LIN {X -0.135,Y -571.189,Z 1193.398,A 0.000,B 0.000,C 90.000,E1 107.583} C_DIS
LIN {X 0.208,Y -571.999,Z 1193.396,A 0.000,B 0.000,C 90.000,E1 107.275} C_DIS
LIN {X -0.181,Y -573.328,Z 1193.392,A 0.000,B 0.000,C 90.000,E1 106.496} C_DIS
LIN {X -0.198,Y -574.045,Z 1193.389,A 0.000,B 0.000,C 90.000,E1 105.953} C_DIS
LIN {X 0.188,Y -574.248,Z 1193.385,A 0.000,B 0.000,C 90.000,E1 105.371} C_DIS
LIN {X 0.176,Y -573.890,Z 1193.383,A 0.000,B 0.000,C 90.000,E1 104.828} C_DIS
LIN {X 0.213,Y -573.031,Z 1193.378,A 0.000,B 0.000,C 90.000,E1 104.008} C_DIS
LIN {X 0.050,Y -571.576,Z 1193.375,A 0.000,B 0.000,C 90.000,E1 103.480} C_DIS
LIN {X 0.009,Y -569.589,Z 1193.372,A 0.000,B 0.000,C 90.000,E1 102.939} C_DIS
LIN {X -0.051,Y -567.766,Z 1193.370,A 0.000,B 0.000,C 90.000,E1 102.535} C_DIS
LIN {X 0.001,Y -565.659,Z 1193.367,A 0.000,B 0.000,C 90.000,E1 102.119} C_DIS
LIN {X -0.053,Y -561.217,Z 1193.363,A 0.000,B 0.000,C 90.000,E1 101.299} C_DIS
LIN {X 0.246,Y -560.479,Z 1193.362,A 0.000,B 0.000,C 90.000,E1 101.130} C_DIS
LIN {X 0.102,Y -560.323,Z 1193.361,A 0.000,B 0.000,C 90.000,E1 101.007} C_DIS
LIN {X -0.002,Y -559.039,Z 1193.359,A 0.000,B 0.000,C 90.000,E1 100.602} C_DIS
LIN {X -0.252,Y -559.123,Z 1193.358,A 0.000,B 0.000,C 90.000,E1 100.489} C_DIS
LIN {X -0.108,Y -558.918,Z 1193.357,A 0.000,B 0.000,C 90.000,E1 100.197} C_DIS
LIN {X 0.289,Y -558.596,Z 1193.356,A 0.000,B 0.000,C 90.000,E1 100.018} C_DIS
LIN {X -0.167,Y -558.552,Z 1193.353,A 0.000,B 0.000,C 90.000,E1 99.500} C_DIS
LIN {X -0.161,Y -560.240,Z 1193.340,A 0.000,B 0.000,C 90.000,E1 97.125} C_DIS
LIN {X -0.058,Y -561.502,Z 1193.330,A 0.000,B 0.000,C 90.000,E1 95.454} C_DIS
LIN {X 0.160,Y -562.825,Z 1193.320,A 0.000,B 0.000,C 90.000,E1 93.498} C_DIS
LIN {X 0.239,Y -563.966,Z 1193.310,A 0.000,B 0.000,C 90.000,E1 91.835} C_DIS
LIN {X -0.224,Y -565.226,Z 1193.301,A 0.000,B 0.000,C 90.000,E1 90.229} C_DIS
LIN {X 0.003,Y -566.586,Z 1193.291,A 0.000,B 0.000,C 90.000,E1 88.282} C_DIS
LIN {X 0.034,Y -567.595,Z 1193.283,A 0.000,B 0.000,C 90.000,E1 86.906} C_DIS
LIN {X 0.234,Y -568.811,Z 1193.274,A 0.000,B 0.000,C 90.000,E1 85.241} C_DIS
LIN {X -0.169,Y -569.801,Z 1193.266,A 0.000,B 0.000,C 90.000,E1 83.913} C_DIS
LIN {X 0.134,Y -570.980,Z 1193.257,A 0.000,B 0.000,C 90.000,E1 82.243} C_DIS
LIN {X -0.140,Y -571.903,Z 1193.249,A 0.000,B 0.000,C 90.000,E1 80.905} C_DIS
LIN {X -0.193,Y -572.866,Z 1193.240,A 0.000,B 0.000,C 90.000,E1 79.275} C_DIS
LIN {X -0.072,Y -573.529,Z 1193.234,A 0.000,B 0.000,C 90.000,E1 78.173} C_DIS
LIN {X -0.194,Y -574.243,Z 1193.227,A 0.000,B 0.000,C 90.000,E1 76.825} C_DIS
LIN {X -0.178,Y -575.213,Z 1193.216,A 0.000,B 0.000,C 90.000,E1 74.921} C_DIS
LIN {X 0.224,Y -575.753,Z 1193.210,A 0.000,B 0.000,C 90.000,E1 73.795} C_DIS
LIN {X -0.273,Y -576.777,Z 1193.200,A 0.000,B 0.000,C 90.000,E1 71.945} C_DIS
LIN {X -0.010,Y -578.184,Z 1193.188,A 0.000,B 0.000,C 90.000,E1 69.752} C_DIS
LIN {X -0.008,Y -580.380,Z 1193.172,A 0.000,B 0.000,C 90.000,E1 67.050} C_DIS
LIN {X 0.359,Y -581.712,Z 1193.165,A 0.000,B 0.000,C 90.000,E1 65.665} C_DIS
LIN {X -0.157,Y -583.727,Z 1193.153,A 0.000,B 0.000,C 90.000,E1 63.563} C_DIS
LIN {X -0.109,Y -585.371,Z 1193.144,A 0.000,B 0.000,C 90.000,E1 61.948} C_DIS
LIN {X 0.082,Y -586.685,Z 1193.137,A 0.000,B 0.000,C 90.000,E1 60.589} C_DIS
LIN {X 0.073,Y -587.872,Z 1193.129,A 0.000,B 0.000,C 90.000,E1 59.253} C_DIS
LIN {X 0.085,Y -588.971,Z 1193.122,A 0.000,B 0.000,C 90.000,E1 57.916} C_DIS
LIN {X 0.106,Y -590.013,Z 1193.114,A 0.000,B 0.000,C 90.000,E1 56.580} C_DIS
LIN {X 0.173,Y -591.189,Z 1193.106,A 0.000,B 0.000,C 90.000,E1 54.975} C_DIS
LIN {X -0.213,Y -592.385,Z 1193.097,A 0.000,B 0.000,C 90.000,E1 53.417} C_DIS
LIN {X -0.002,Y -593.609,Z 1193.086,A 0.000,B 0.000,C 90.000,E1 51.537} C_DIS
LIN {X 0.170,Y -594.350,Z 1193.079,A 0.000,B 0.000,C 90.000,E1 50.194} C_DIS
LIN {X 0.354,Y -595.043,Z 1193.072,A 0.000,B 0.000,C 90.000,E1 48.852} C_DIS
LIN {X 0.095,Y -595.432,Z 1193.064,A 0.000,B 0.000,C 90.000,E1 47.553} C_DIS
LIN {X -0.149,Y -595.602,Z 1193.060,A 0.000,B 0.000,C 90.000,E1 46.782} C_DIS
LIN {X -0.205,Y -595.657,Z 1193.054,A 0.000,B 0.000,C 90.000,E1 45.729} C_DIS
LIN {X -0.256,Y -595.587,Z 1193.048,A 0.000,B 0.000,C 90.000,E1 44.676} C_DIS
LIN {X -0.310,Y -595.335,Z 1193.042,A 0.000,B 0.000,C 90.000,E1 43.623} C_DIS
LIN {X 0.288,Y -594.985,Z 1193.038,A 0.000,B 0.000,C 90.000,E1 42.771} C_DIS
LIN {X -0.187,Y -594.334,Z 1193.032,A 0.000,B 0.000,C 90.000,E1 41.757} C_DIS
LIN {X -0.011,Y -593.310,Z 1193.025,A 0.000,B 0.000,C 90.000,E1 40.415} C_DIS
LIN {X -0.034,Y -592.965,Z 1193.022,A 0.000,B 0.000,C 90.000,E1 39.886} C_DIS
LIN {X -0.092,Y -591.934,Z 1193.016,A 0.000,B 0.000,C 90.000,E1 38.830} C_DIS
LIN {X 0.289,Y -590.732,Z 1193.010,A 0.000,B 0.000,C 90.000,E1 37.729} C_DIS
LIN {X -0.178,Y -589.270,Z 1193.004,A 0.000,B 0.000,C 90.000,E1 36.710} C_DIS
LIN {X 0.281,Y -587.627,Z 1192.998,A 0.000,B 0.000,C 90.000,E1 35.598} C_DIS
LIN {X 0.095,Y -584.955,Z 1192.990,A 0.000,B 0.000,C 90.000,E1 34.278} C_DIS
LIN {X -0.347,Y -583.610,Z 1192.988,A 0.000,B 0.000,C 90.000,E1 33.785} C_DIS
LIN {X 0.031,Y -580.538,Z 1192.982,A 0.000,B 0.000,C 90.000,E1 32.673} C_DIS
LIN {X 0.043,Y -578.829,Z 1192.979,A 0.000,B 0.000,C 90.000,E1 32.133} C_DIS
LIN {X 0.044,Y -576.919,Z 1192.976,A 0.000,B 0.000,C 90.000,E1 31.592} C_DIS
LIN {X 0.003,Y -572.581,Z 1192.970,A 0.000,B 0.000,C 90.000,E1 30.512} C_DIS
LIN {X 0.276,Y -568.708,Z 1192.965,A 0.000,B 0.000,C 90.000,E1 29.667} C_DIS
LIN {X 0.010,Y -566.668,Z 1192.963,A 0.000,B 0.000,C 90.000,E1 29.283} C_DIS
LIN {X -0.175,Y -562.965,Z 1192.959,A 0.000,B 0.000,C 90.000,E1 28.615} C_DIS
LIN {X 0.197,Y -559.863,Z 1192.956,A 0.000,B 0.000,C 90.000,E1 28.025} C_DIS
LIN {X 0.179,Y -555.637,Z 1192.952,A 0.000,B 0.000,C 90.000,E1 27.334} C_DIS
LIN {X 0.266,Y -550.248,Z 1192.947,A 0.000,B 0.000,C 90.000,E1 26.488} C_DIS
LIN {X -0.200,Y -546.283,Z 1192.944,A 0.000,B 0.000,C 90.000,E1 25.976} C_DIS
LIN {X -0.099,Y -542.123,Z 1192.941,A 0.000,B 0.000,C 90.000,E1 25.412} C_DIS
LIN {X -0.033,Y -536.403,Z 1192.937,A 0.000,B 0.000,C 90.000,E1 24.695} C_DIS
LIN {X 0.237,Y -530.425,Z 1192.933,A 0.000,B 0.000,C 90.000,E1 23.951} C_DIS
LIN {X -0.025,Y -523.948,Z 1192.929,A 0.000,B 0.000,C 90.000,E1 23.259} C_DIS
LIN {X -0.185,Y -516.325,Z 1192.925,A 0.000,B 0.000,C 90.000,E1 22.461} C_DIS
LIN {X 0.185,Y -506.933,Z 1192.919,A 0.000,B 0.000,C 90.000,E1 21.461} C_DIS
LIN {X 0.093,Y -499.911,Z 1192.916,A 0.000,B 0.000,C 90.000,E1 20.791} C_DIS
LIN {X 0.041,Y -492.746,Z 1192.912,A 0.000,B 0.000,C 90.000,E1 20.120} C_DIS
LIN {X 0.132,Y -484.080,Z 1192.907,A 0.000,B 0.000,C 90.000,E1 19.322} C_DIS
LIN {X 0.217,Y -475.597,Z 1192.903,A 0.000,B 0.000,C 90.000,E1 18.544} C_DIS
LIN {X -0.018,Y -468.551,Z 1192.900,A 0.000,B 0.000,C 90.000,E1 17.946} C_DIS
LIN {X -0.152,Y -449.674,Z 1192.890,A 0.000,B 0.000,C 90.000,E1 16.260} C_DIS
LIN {X -0.141,Y -427.913,Z 1192.878,A 0.000,B 0.000,C 90.000,E1 14.120} C_DIS
LIN {X 0.092,Y -413.875,Z 1192.870,A 0.000,B 0.000,C 90.000,E1 12.535} C_DIS
LIN {X -0.060,Y -403.114,Z 1192.862,A 0.000,B 0.000,C 90.000,E1 11.243} C_DIS
LIN {X -0.062,Y -398.061,Z 1192.859,A 0.000,B 0.000,C 90.000,E1 10.546} C_DIS
LIN {X -0.007,Y -395.199,Z 1192.856,A 0.000,B 0.000,C 90.000,E1 10.074} C_DIS
LIN {X -0.001,Y -393.528,Z 1192.854,A 0.000,B 0.000,C 90.000,E1 9.670} C_DIS
LIN {X -0.038,Y -393.515,Z 1192.854,A 0.000,B 0.000,C 90.000,E1 9.670} C_DIS
LIN {X -0.114,Y -393.293,Z 1192.852,A 0.000,B 0.000,C 90.000,E1 9.321} C_DIS
LIN {X -0.152,Y -393.295,Z 1192.852,A 0.000,B 0.000,C 90.000,E1 9.321} C_DIS
LIN {X -0.137,Y -394.226,Z 1192.849,A 0.000,B 0.000,C 90.000,E1 8.859} C_DIS
LIN {X 0.180,Y -396.841,Z 1192.845,A 0.000,B 0.000,C 90.000,E1 8.106} C_DIS
LIN {X 0.138,Y -397.747,Z 1192.844,A 0.000,B 0.000,C 90.000,E1 7.936} C_DIS
LIN {X 0.094,Y -402.181,Z 1192.840,A 0.000,B 0.000,C 90.000,E1 7.239} C_DIS
LIN {X -0.167,Y -406.787,Z 1192.838,A 0.000,B 0.000,C 90.000,E1 6.777} C_DIS
LIN {X -0.181,Y -412.209,Z 1192.835,A 0.000,B 0.000,C 90.000,E1 6.315} C_DIS
LIN {X -0.046,Y -426.154,Z 1192.829,A 0.000,B 0.000,C 90.000,E1 5.220} C_DIS
LIN {X 0.015,Y -438.945,Z 1192.824,A 0.000,B 0.000,C 90.000,E1 4.245} C_DIS
LIN {X -0.229,Y -453.424,Z 1192.818,A 0.000,B 0.000,C 90.000,E1 3.212} C_DIS
LIN {X -0.129,Y -465.940,Z 1192.813,A 0.000,B 0.000,C 90.000,E1 2.293} C_DIS
LIN {X 0.221,Y -475.191,Z 1192.809,A 0.000,B 0.000,C 90.000,E1 1.547} C_DIS
LIN {X -0.118,Y -484.281,Z 1192.805,A 0.000,B 0.000,C 90.000,E1 0.859} C_DIS
LIN {X 0.099,Y -491.240,Z 1192.801,A 0.000,B 0.000,C 90.000,E1 0.229} C_DIS
LIN {X 0.013,Y -497.431,Z 1192.798,A 0.000,B 0.000,C 90.000,E1 359.656} C_DIS
LIN {X 0.078,Y -504.088,Z 1192.794,A 0.000,B 0.000,C 90.000,E1 358.969} C_DIS
LIN {X -0.006,Y -511.739,Z 1192.790,A 0.000,B 0.000,C 90.000,E1 358.108} C_DIS
LIN {X -0.173,Y -516.632,Z 1192.786,A 0.000,B 0.000,C 90.000,E1 357.535} C_DIS
LIN {X -0.052,Y -522.198,Z 1192.782,A 0.000,B 0.000,C 90.000,E1 356.788} C_DIS
LIN {X 0.089,Y -527.295,Z 1192.778,A 0.000,B 0.000,C 90.000,E1 356.045} C_DIS
LIN {X 0.059,Y -531.040,Z 1192.775,A 0.000,B 0.000,C 90.000,E1 355.469} C_DIS
LIN {X -0.215,Y -535.271,Z 1192.771,A 0.000,B 0.000,C 90.000,E1 354.780} C_DIS
LIN {X 0.078,Y -539.012,Z 1192.767,A 0.000,B 0.000,C 90.000,E1 354.033} C_DIS
LIN {X -0.069,Y -542.455,Z 1192.763,A 0.000,B 0.000,C 90.000,E1 353.337} C_DIS
LIN {X -0.251,Y -545.552,Z 1192.759,A 0.000,B 0.000,C 90.000,E1 352.648} C_DIS
LIN {X -0.061,Y -548.907,Z 1192.754,A 0.000,B 0.000,C 90.000,E1 351.781} C_DIS
LIN {X 0.251,Y -551.963,Z 1192.750,A 0.000,B 0.000,C 90.000,E1 350.905} C_DIS
LIN {X 0.092,Y -555.560,Z 1192.743,A 0.000,B 0.000,C 90.000,E1 349.803} C_DIS
LIN {X -0.027,Y -558.720,Z 1192.737,A 0.000,B 0.000,C 90.000,E1 348.701} C_DIS
LIN {X 0.001,Y -561.616,Z 1192.731,A 0.000,B 0.000,C 90.000,E1 347.589} C_DIS
LIN {X 0.199,Y -564.253,Z 1192.725,A 0.000,B 0.000,C 90.000,E1 346.464} C_DIS
LIN {X 0.065,Y -567.321,Z 1192.717,A 0.000,B 0.000,C 90.000,E1 345.102} C_DIS
LIN {X -0.194,Y -569.642,Z 1192.711,A 0.000,B 0.000,C 90.000,E1 344.031} C_DIS
LIN {X 0.099,Y -572.817,Z 1192.702,A 0.000,B 0.000,C 90.000,E1 342.362} C_DIS
LIN {X -0.288,Y -575.201,Z 1192.695,A 0.000,B 0.000,C 90.000,E1 341.040} C_DIS
LIN {X -0.085,Y -576.829,Z 1192.688,A 0.000,B 0.000,C 90.000,E1 339.934} C_DIS
LIN {X -0.216,Y -578.505,Z 1192.681,A 0.000,B 0.000,C 90.000,E1 338.592} C_DIS
LIN {X 0.035,Y -579.400,Z 1192.675,A 0.000,B 0.000,C 90.000,E1 337.486} C_DIS
LIN {X 0.277,Y -579.714,Z 1192.672,A 0.000,B 0.000,C 90.000,E1 336.922} C_DIS
LIN {X 0.147,Y -579.928,Z 1192.667,A 0.000,B 0.000,C 90.000,E1 336.125} C_DIS
LIN {X 0.108,Y -579.665,Z 1192.661,A 0.000,B 0.000,C 90.000,E1 335.049} C_DIS
LIN {X -0.173,Y -579.328,Z 1192.658,A 0.000,B 0.000,C 90.000,E1 334.537} C_DIS
LIN {X -0.076,Y -578.494,Z 1192.654,A 0.000,B 0.000,C 90.000,E1 333.717} C_DIS
LIN {X 0.269,Y -577.267,Z 1192.650,A 0.000,B 0.000,C 90.000,E1 332.871} C_DIS
LIN {X -0.174,Y -575.623,Z 1192.645,A 0.000,B 0.000,C 90.000,E1 332.103} C_DIS
LIN {X 0.143,Y -573.696,Z 1192.641,A 0.000,B 0.000,C 90.000,E1 331.257} C_DIS
LIN {X -0.062,Y -571.446,Z 1192.636,A 0.000,B 0.000,C 90.000,E1 330.461} C_DIS
LIN {X -0.114,Y -569.543,Z 1192.633,A 0.000,B 0.000,C 90.000,E1 329.921} C_DIS
LIN {X 0.115,Y -567.902,Z 1192.631,A 0.000,B 0.000,C 90.000,E1 329.488} C_DIS
LIN {X 0.036,Y -565.377,Z 1192.628,A 0.000,B 0.000,C 90.000,E1 328.948} C_DIS
LIN {X -0.059,Y -562.440,Z 1192.625,A 0.000,B 0.000,C 90.000,E1 328.408} C_DIS
LIN {X 0.019,Y -558.086,Z 1192.621,A 0.000,B 0.000,C 90.000,E1 327.709} C_DIS
LIN {X -0.052,Y -552.201,Z 1192.616,A 0.000,B 0.000,C 90.000,E1 326.882} C_DIS
LIN {X 0.348,Y -549.045,Z 1192.614,A 0.000,B 0.000,C 90.000,E1 326.421} C_DIS
LIN {X 0.005,Y -543.342,Z 1192.610,A 0.000,B 0.000,C 90.000,E1 325.754} C_DIS
LIN {X 0.078,Y -536.190,Z 1192.605,A 0.000,B 0.000,C 90.000,E1 324.895} C_DIS
LIN {X -0.066,Y -529.931,Z 1192.601,A 0.000,B 0.000,C 90.000,E1 324.196} C_DIS
LIN {X -0.238,Y -523.645,Z 1192.597,A 0.000,B 0.000,C 90.000,E1 323.497} C_DIS
LIN {X 0.144,Y -519.570,Z 1192.594,A 0.000,B 0.000,C 90.000,E1 322.924} C_DIS
LIN {X 0.251,Y -517.243,Z 1192.592,A 0.000,B 0.000,C 90.000,E1 322.557} C_DIS
LIN {X -0.102,Y -514.817,Z 1192.589,A 0.000,B 0.000,C 90.000,E1 322.110} C_DIS
LIN {X 0.056,Y -513.874,Z 1192.588,A 0.000,B 0.000,C 90.000,E1 321.778} C_DIS
LIN {X -0.019,Y -513.107,Z 1192.586,A 0.000,B 0.000,C 90.000,E1 321.492} C_DIS
LIN {X 0.146,Y -512.472,Z 1192.583,A 0.000,B 0.000,C 90.000,E1 320.884} C_DIS
LIN {X -0.019,Y -512.285,Z 1192.580,A 0.000,B 0.000,C 90.000,E1 320.312} C_DIS
LIN {X 0.166,Y -513.720,Z 1192.565,A 0.000,B 0.000,C 90.000,E1 317.634} C_DIS
LIN {X 0.132,Y -514.389,Z 1192.558,A 0.000,B 0.000,C 90.000,E1 316.458} C_DIS
LIN {X 0.083,Y -515.713,Z 1192.545,A 0.000,B 0.000,C 90.000,E1 314.109} C_DIS
LIN {X 0.353,Y -516.532,Z 1192.537,A 0.000,B 0.000,C 90.000,E1 312.609} C_DIS
LIN {X -0.171,Y -517.686,Z 1192.527,A 0.000,B 0.000,C 90.000,E1 310.906} C_DIS
LIN {X -0.034,Y -518.229,Z 1192.522,A 0.000,B 0.000,C 90.000,E1 310.011} C_DIS
LIN {X -0.064,Y -519.313,Z 1192.513,A 0.000,B 0.000,C 90.000,E1 308.257} C_DIS
LIN {X -0.021,Y -520.105,Z 1192.504,A 0.000,B 0.000,C 90.000,E1 306.790} C_DIS
LIN {X 0.139,Y -520.852,Z 1192.496,A 0.000,B 0.000,C 90.000,E1 305.311} C_DIS
LIN {X -0.082,Y -521.822,Z 1192.485,A 0.000,B 0.000,C 90.000,E1 303.293} C_DIS
LIN {X -0.138,Y -522.384,Z 1192.479,A 0.000,B 0.000,C 90.000,E1 302.133} C_DIS
LIN {X -0.069,Y -522.959,Z 1192.470,A 0.000,B 0.000,C 90.000,E1 300.669} C_DIS
LIN {X 0.075,Y -523.270,Z 1192.464,A 0.000,B 0.000,C 90.000,E1 299.489} C_DIS
LIN {X -0.161,Y -523.634,Z 1192.454,A 0.000,B 0.000,C 90.000,E1 297.769} C_DIS
LIN {X 0.284,Y -523.855,Z 1192.445,A 0.000,B 0.000,C 90.000,E1 295.976} C_DIS
LIN {X -0.128,Y -523.920,Z 1192.436,A 0.000,B 0.000,C 90.000,E1 294.567} C_DIS
LIN {X -0.125,Y -523.759,Z 1192.427,A 0.000,B 0.000,C 90.000,E1 292.823} C_DIS
LIN {X -0.158,Y -523.694,Z 1192.415,A 0.000,B 0.000,C 90.000,E1 290.791} C_DIS
LIN {X -0.042,Y -523.539,Z 1192.406,A 0.000,B 0.000,C 90.000,E1 289.033} C_DIS
LIN {X -0.076,Y -523.090,Z 1192.399,A 0.000,B 0.000,C 90.000,E1 287.873} C_DIS
LIN {X -0.288,Y -522.444,Z 1192.391,A 0.000,B 0.000,C 90.000,E1 286.441} C_DIS
LIN {X -0.006,Y -521.731,Z 1192.385,A 0.000,B 0.000,C 90.000,E1 285.245} C_DIS
LIN {X 0.127,Y -520.731,Z 1192.377,A 0.000,B 0.000,C 90.000,E1 283.772} C_DIS
LIN {X 0.240,Y -519.307,Z 1192.365,A 0.000,B 0.000,C 90.000,E1 281.715} C_DIS
LIN {X 0.220,Y -518.418,Z 1192.357,A 0.000,B 0.000,C 90.000,E1 280.254} C_DIS
LIN {X 0.081,Y -517.480,Z 1192.347,A 0.000,B 0.000,C 90.000,E1 278.511} C_DIS
LIN {X -0.178,Y -516.429,Z 1192.336,A 0.000,B 0.000,C 90.000,E1 276.486} C_DIS
LIN {X 0.009,Y -515.343,Z 1192.326,A 0.000,B 0.000,C 90.000,E1 274.702} C_DIS
LIN {X -0.094,Y -513.855,Z 1192.311,A 0.000,B 0.000,C 90.000,E1 272.064} C_DIS
LIN {X 0.056,Y -513.164,Z 1192.303,A 0.000,B 0.000,C 90.000,E1 270.573} C_DIS
LIN {X 0.180,Y -512.445,Z 1192.295,A 0.000,B 0.000,C 90.000,E1 269.083} C_DIS
LIN {X -0.062,Y -511.959,Z 1192.290,A 0.000,B 0.000,C 90.000,E1 268.224} C_DIS
LIN {X -0.016,Y -510.835,Z 1192.280,A 0.000,B 0.000,C 90.000,E1 266.445} C_DIS
LIN {X 0.105,Y -509.755,Z 1192.272,A 0.000,B 0.000,C 90.000,E1 264.951} C_DIS
LIN {X 0.146,Y -507.991,Z 1192.262,A 0.000,B 0.000,C 90.000,E1 263.166} C_DIS
LIN {X 0.201,Y -506.433,Z 1192.252,A 0.000,B 0.000,C 90.000,E1 261.376} C_DIS
LIN {X -0.262,Y -504.757,Z 1192.241,A 0.000,B 0.000,C 90.000,E1 259.342} C_DIS
LIN {X 0.001,Y -503.693,Z 1192.234,A 0.000,B 0.000,C 90.000,E1 258.117} C_DIS
LIN {X -0.136,Y -502.728,Z 1192.227,A 0.000,B 0.000,C 90.000,E1 256.937} C_DIS
LIN {X 0.191,Y -501.237,Z 1192.217,A 0.000,B 0.000,C 90.000,E1 255.102} C_DIS
LIN {X 0.028,Y -499.184,Z 1192.202,A 0.000,B 0.000,C 90.000,E1 252.417} C_DIS
LIN {X -0.041,Y -498.354,Z 1192.196,A 0.000,B 0.000,C 90.000,E1 251.221} C_DIS
LIN {X 0.205,Y -496.514,Z 1192.184,A 0.000,B 0.000,C 90.000,E1 249.082} C_DIS
LIN {X 0.075,Y -494.857,Z 1192.174,A 0.000,B 0.000,C 90.000,E1 247.283} C_DIS
LIN {X -0.137,Y -493.344,Z 1192.166,A 0.000,B 0.000,C 90.000,E1 245.793} C_DIS
LIN {X 0.191,Y -492.498,Z 1192.160,A 0.000,B 0.000,C 90.000,E1 244.845} C_DIS
LIN {X -0.069,Y -490.339,Z 1192.150,A 0.000,B 0.000,C 90.000,E1 243.050} C_DIS
LIN {X 0.028,Y -488.871,Z 1192.144,A 0.000,B 0.000,C 90.000,E1 241.820} C_DIS
LIN {X -0.088,Y -486.517,Z 1192.133,A 0.000,B 0.000,C 90.000,E1 239.999} C_DIS
LIN {X -0.005,Y -484.573,Z 1192.125,A 0.000,B 0.000,C 90.000,E1 238.456} C_DIS
LIN {X 0.038,Y -482.580,Z 1192.116,A 0.000,B 0.000,C 90.000,E1 236.914} C_DIS
LIN {X -0.090,Y -479.738,Z 1192.104,A 0.000,B 0.000,C 90.000,E1 234.769} C_DIS
LIN {X -0.204,Y -477.423,Z 1192.094,A 0.000,B 0.000,C 90.000,E1 232.924} C_DIS
LIN {X -0.209,Y -474.326,Z 1192.080,A 0.000,B 0.000,C 90.000,E1 230.436} C_DIS
LIN {X -0.010,Y -472.421,Z 1192.071,A 0.000,B 0.000,C 90.000,E1 228.852} C_DIS
LIN {X -0.202,Y -470.417,Z 1192.063,A 0.000,B 0.000,C 90.000,E1 227.310} C_DIS
LIN {X 0.265,Y -466.769,Z 1192.045,A 0.000,B 0.000,C 90.000,E1 224.109} C_DIS
LIN {X 0.152,Y -464.568,Z 1192.031,A 0.000,B 0.000,C 90.000,E1 221.595} C_DIS
LIN {X 0.271,Y -463.522,Z 1192.012,A 0.000,B 0.000,C 90.000,E1 218.096} C_DIS
LIN {X 0.179,Y -463.573,Z 1192.007,A 0.000,B 0.000,C 90.000,E1 217.156} C_DIS
LIN {X -0.034,Y -463.600,Z 1191.998,A 0.000,B 0.000,C 90.000,E1 215.598} C_DIS
LIN {X -0.116,Y -463.891,Z 1191.987,A 0.000,B 0.000,C 90.000,E1 213.706} C_DIS
LIN {X 0.025,Y -466.201,Z 1191.968,A 0.000,B 0.000,C 90.000,E1 210.207} C_DIS
LIN {X -0.108,Y -469.064,Z 1191.952,A 0.000,B 0.000,C 90.000,E1 207.385} C_DIS
LIN {X 0.037,Y -470.778,Z 1191.943,A 0.000,B 0.000,C 90.000,E1 205.796} C_DIS
LIN {X 0.088,Y -478.976,Z 1191.914,A 0.000,B 0.000,C 90.000,E1 200.482} C_DIS
LIN {X 0.028,Y -486.617,Z 1191.895,A 0.000,B 0.000,C 90.000,E1 197.094} C_DIS
LIN {X -0.073,Y -493.324,Z 1191.881,A 0.000,B 0.000,C 90.000,E1 194.662} C_DIS
LIN {X 0.165,Y -497.843,Z 1191.873,A 0.000,B 0.000,C 90.000,E1 193.119} C_DIS
LIN {X 0.233,Y -504.410,Z 1191.861,A 0.000,B 0.000,C 90.000,E1 191.007} C_DIS
LIN {X 0.245,Y -512.287,Z 1191.848,A 0.000,B 0.000,C 90.000,E1 188.624} C_DIS
LIN {X -0.049,Y -517.219,Z 1191.840,A 0.000,B 0.000,C 90.000,E1 187.182} C_DIS
LIN {X -0.185,Y -521.118,Z 1191.833,A 0.000,B 0.000,C 90.000,E1 186.024} C_DIS
LIN {X 0.103,Y -527.883,Z 1191.822,A 0.000,B 0.000,C 90.000,E1 183.955} C_DIS
LIN {X 0.023,Y -531.715,Z 1191.816,A 0.000,B 0.000,C 90.000,E1 182.808} C_DIS
LIN {X -0.005,Y -536.525,Z 1191.808,A 0.000,B 0.000,C 90.000,E1 181.375} C_DIS
LIN {X 0.089,Y -543.214,Z 1191.797,A 0.000,B 0.000,C 90.000,E1 179.370} C_DIS
LIN {X -0.183,Y -549.820,Z 1191.786,A 0.000,B 0.000,C 90.000,E1 177.421} C_DIS
LIN {X 0.118,Y -554.447,Z 1191.778,A 0.000,B 0.000,C 90.000,E1 175.988} C_DIS
LIN {X -0.088,Y -558.087,Z 1191.772,A 0.000,B 0.000,C 90.000,E1 174.894} C_DIS
LIN {X -0.015,Y -563.444,Z 1191.762,A 0.000,B 0.000,C 90.000,E1 173.223} C_DIS
LIN {X 0.244,Y -568.733,Z 1191.753,A 0.000,B 0.000,C 90.000,E1 171.546} C_DIS
LIN {X 0.045,Y -573.895,Z 1191.744,A 0.000,B 0.000,C 90.000,E1 169.926} C_DIS
LIN {X 0.292,Y -577.287,Z 1191.738,A 0.000,B 0.000,C 90.000,E1 168.814} C_DIS
LIN {X -0.084,Y -582.463,Z 1191.729,A 0.000,B 0.000,C 90.000,E1 167.229} C_DIS
LIN {X 0.206,Y -587.564,Z 1191.720,A 0.000,B 0.000,C 90.000,E1 165.589} C_DIS
LIN {X -0.034,Y -590.128,Z 1191.716,A 0.000,B 0.000,C 90.000,E1 164.810} C_DIS
LIN {X -0.153,Y -596.051,Z 1191.705,A 0.000,B 0.000,C 90.000,E1 162.960} C_DIS
LIN {X 0.143,Y -601.144,Z 1191.697,A 0.000,B 0.000,C 90.000,E1 161.348} C_DIS
LIN {X 0.366,Y -606.095,Z 1191.688,A 0.000,B 0.000,C 90.000,E1 159.752} C_DIS
LIN {X 0.190,Y -610.202,Z 1191.681,A 0.000,B 0.000,C 90.000,E1 158.465} C_DIS
LIN {X 0.011,Y -615.864,Z 1191.670,A 0.000,B 0.000,C 90.000,E1 156.666} C_DIS
LIN {X 0.227,Y -619.782,Z 1191.663,A 0.000,B 0.000,C 90.000,E1 155.357} C_DIS
LIN {X -0.064,Y -623.609,Z 1191.656,A 0.000,B 0.000,C 90.000,E1 154.101} C_DIS
LIN {X -0.026,Y -627.250,Z 1191.649,A 0.000,B 0.000,C 90.000,E1 152.820} C_DIS
LIN {X -0.189,Y -630.795,Z 1191.642,A 0.000,B 0.000,C 90.000,E1 151.563} C_DIS
LIN {X 0.312,Y -634.894,Z 1191.634,A 0.000,B 0.000,C 90.000,E1 149.999} C_DIS
LIN {X 0.288,Y -638.086,Z 1191.627,A 0.000,B 0.000,C 90.000,E1 148.742} C_DIS
LIN {X -0.237,Y -641.107,Z 1191.620,A 0.000,B 0.000,C 90.000,E1 147.533} C_DIS
LIN {X -0.370,Y -643.941,Z 1191.613,A 0.000,B 0.000,C 90.000,E1 146.294} C_DIS
LIN {X -0.036,Y -647.084,Z 1191.604,A 0.000,B 0.000,C 90.000,E1 144.769} C_DIS
LIN {X -0.223,Y -649.440,Z 1191.597,A 0.000,B 0.000,C 90.000,E1 143.543} C_DIS
LIN {X 0.085,Y -652.241,Z 1191.589,A 0.000,B 0.000,C 90.000,E1 142.029} C_DIS
LIN {X -0.079,Y -655.988,Z 1191.578,A 0.000,B 0.000,C 90.000,E1 140.070} C_DIS
LIN {X -0.175,Y -657.992,Z 1191.573,A 0.000,B 0.000,C 90.000,E1 139.094} C_DIS
LIN {X -0.323,Y -661.673,Z 1191.563,A 0.000,B 0.000,C 90.000,E1 137.391} C_DIS
LIN {X 0.077,Y -664.769,Z 1191.555,A 0.000,B 0.000,C 90.000,E1 135.891} C_DIS
LIN {X 0.078,Y -669.637,Z 1191.543,A 0.000,B 0.000,C 90.000,E1 133.704} C_DIS
LIN {X 0.204,Y -673.672,Z 1191.533,A 0.000,B 0.000,C 90.000,E1 132.000} C_DIS
LIN {X -0.165,Y -675.994,Z 1191.528,A 0.000,B 0.000,C 90.000,E1 131.067} C_DIS
LIN {X 0.204,Y -680.728,Z 1191.517,A 0.000,B 0.000,C 90.000,E1 129.116} C_DIS
LIN {X 0.224,Y -684.872,Z 1191.508,A 0.000,B 0.000,C 90.000,E1 127.443} C_DIS
LIN {X -0.296,Y -687.857,Z 1191.502,A 0.000,B 0.000,C 90.000,E1 126.297} C_DIS
LIN {X 0.151,Y -690.219,Z 1191.496,A 0.000,B 0.000,C 90.000,E1 125.311} C_DIS
LIN {X 0.167,Y -694.578,Z 1191.486,A 0.000,B 0.000,C 90.000,E1 123.420} C_DIS
LIN {X -0.036,Y -697.120,Z 1191.479,A 0.000,B 0.000,C 90.000,E1 122.260} C_DIS
LIN {X -0.228,Y -699.064,Z 1191.474,A 0.000,B 0.000,C 90.000,E1 121.337} C_DIS
LIN {X -0.031,Y -700.891,Z 1191.469,A 0.000,B 0.000,C 90.000,E1 120.384} C_DIS
LIN {X -0.172,Y -702.541,Z 1191.464,A 0.000,B 0.000,C 90.000,E1 119.461} C_DIS
LIN {X -0.012,Y -704.413,Z 1191.457,A 0.000,B 0.000,C 90.000,E1 118.281} C_DIS
LIN {X -0.107,Y -705.400,Z 1191.453,A 0.000,B 0.000,C 90.000,E1 117.590} C_DIS
LIN {X 0.139,Y -706.091,Z 1191.449,A 0.000,B 0.000,C 90.000,E1 116.873} C_DIS
LIN {X -0.268,Y -706.595,Z 1191.444,A 0.000,B 0.000,C 90.000,E1 115.976} C_DIS
LIN {X 0.321,Y -706.710,Z 1191.442,A 0.000,B 0.000,C 90.000,E1 115.463} C_DIS
LIN {X -0.032,Y -706.688,Z 1191.439,A 0.000,B 0.000,C 90.000,E1 115.027} C_DIS
LIN {X -0.088,Y -706.426,Z 1191.437,A 0.000,B 0.000,C 90.000,E1 114.567} C_DIS
LIN {X 0.204,Y -705.577,Z 1191.434,A 0.000,B 0.000,C 90.000,E1 114.079} C_DIS
LIN {X -0.152,Y -705.023,Z 1191.433,A 0.000,B 0.000,C 90.000,E1 113.875} C_DIS
LIN {X 0.274,Y -702.214,Z 1191.429,A 0.000,B 0.000,C 90.000,E1 113.259} C_DIS
LIN {X 0.136,Y -701.307,Z 1191.429,A 0.000,B 0.000,C 90.000,E1 113.153} C_DIS
LIN {X -0.057,Y -696.079,Z 1191.426,A 0.000,B 0.000,C 90.000,E1 112.717} C_DIS
LIN {X 0.175,Y -694.503,Z 1191.426,A 0.000,B 0.000,C 90.000,E1 112.589} C_DIS
LIN {X -0.234,Y -691.698,Z 1191.425,A 0.000,B 0.000,C 90.000,E1 112.514} C_DIS
LIN {X -0.239,Y -685.705,Z 1191.424,A 0.000,B 0.000,C 90.000,E1 112.333} C_DIS
LIN {X 0.155,Y -684.400,Z 1191.424,A 0.000,B 0.000,C 90.000,E1 112.280} C_DIS
LIN {X -0.213,Y -677.137,Z 1191.424,A 0.000,B 0.000,C 90.000,E1 112.280} C_DIS
LIN {X -0.237,Y -607.012,Z 1191.424,A 0.000,B 0.000,C 90.000,E1 112.280} C_DIS
LIN {X -0.160,Y -602.447,Z 1191.422,A 0.000,B 0.000,C 90.000,E1 111.972} C_DIS
LIN {X -0.234,Y -590.877,Z 1191.417,A 0.000,B 0.000,C 90.000,E1 111.046} C_DIS
LIN {X -0.065,Y -580.724,Z 1191.412,A 0.000,B 0.000,C 90.000,E1 110.248} C_DIS
LIN {X -0.026,Y -571.921,Z 1191.409,A 0.000,B 0.000,C 90.000,E1 109.577} C_DIS
LIN {X 0.117,Y -568.925,Z 1191.408,A 0.000,B 0.000,C 90.000,E1 109.341} C_DIS
LIN {X 0.212,Y -565.256,Z 1191.406,A 0.000,B 0.000,C 90.000,E1 109.033} C_DIS
LIN {X -0.201,Y -563.737,Z 1191.405,A 0.000,B 0.000,C 90.000,E1 108.960} C_DIS
LIN {X 0.204,Y -562.542,Z 1191.405,A 0.000,B 0.000,C 90.000,E1 108.779} C_DIS
LIN {X 0.169,Y -562.514,Z 1191.404,A 0.000,B 0.000,C 90.000,E1 108.779} C_DIS
LIN {X 0.170,Y -562.657,Z 1191.402,A 0.000,B 0.000,C 90.000,E1 108.417} C_DIS
LIN {X -0.117,Y -562.825,Z 1191.402,A 0.000,B 0.000,C 90.000,E1 108.308} C_DIS
LIN {X -0.227,Y -567.021,Z 1191.393,A 0.000,B 0.000,C 90.000,E1 106.804} C_DIS
LIN {X -0.285,Y -568.077,Z 1191.390,A 0.000,B 0.000,C 90.000,E1 106.260} C_DIS
LIN {X 0.209,Y -568.163,Z 1191.387,A 0.000,B 0.000,C 90.000,E1 105.662} C_DIS
LIN {X 0.327,Y -567.856,Z 1191.383,A 0.000,B 0.000,C 90.000,E1 104.828} C_DIS
LIN {X 0.125,Y -567.066,Z 1191.380,A 0.000,B 0.000,C 90.000,E1 104.300} C_DIS
LIN {X -0.252,Y -566.394,Z 1191.378,A 0.000,B 0.000,C 90.000,E1 104.064} C_DIS
LIN {X 0.093,Y -564.583,Z 1191.375,A 0.000,B 0.000,C 90.000,E1 103.480} C_DIS
LIN {X -0.158,Y -563.503,Z 1191.373,A 0.000,B 0.000,C 90.000,E1 103.231} C_DIS
LIN {X 0.005,Y -562.610,Z 1191.372,A 0.000,B 0.000,C 90.000,E1 102.939} C_DIS
LIN {X -0.227,Y -560.375,Z 1191.369,A 0.000,B 0.000,C 90.000,E1 102.411} C_DIS
LIN {X 0.214,Y -558.411,Z 1191.367,A 0.000,B 0.000,C 90.000,E1 101.951} C_DIS
LIN {X 0.072,Y -558.180,Z 1191.366,A 0.000,B 0.000,C 90.000,E1 101.827} C_DIS
LIN {X 0.214,Y -557.469,Z 1191.364,A 0.000,B 0.000,C 90.000,E1 101.535} C_DIS
LIN {X 0.025,Y -557.418,Z 1191.360,A 0.000,B 0.000,C 90.000,E1 100.838} C_DIS
LIN {X 0.165,Y -557.647,Z 1191.359,A 0.000,B 0.000,C 90.000,E1 100.546} C_DIS
LIN {X 0.076,Y -560.267,Z 1191.339,A 0.000,B 0.000,C 90.000,E1 96.947} C_DIS
LIN {X 0.169,Y -561.558,Z 1191.329,A 0.000,B 0.000,C 90.000,E1 95.277} C_DIS
LIN {X -0.091,Y -563.024,Z 1191.317,A 0.000,B 0.000,C 90.000,E1 93.094} C_DIS
LIN {X -0.123,Y -564.000,Z 1191.310,A 0.000,B 0.000,C 90.000,E1 91.718} C_DIS
LIN {X -0.038,Y -565.265,Z 1191.300,A 0.000,B 0.000,C 90.000,E1 90.057} C_DIS
LIN {X -0.243,Y -566.814,Z 1191.288,A 0.000,B 0.000,C 90.000,E1 87.879} C_DIS
LIN {X 0.250,Y -567.613,Z 1191.282,A 0.000,B 0.000,C 90.000,E1 86.731} C_DIS
LIN {X -0.104,Y -568.814,Z 1191.273,A 0.000,B 0.000,C 90.000,E1 85.122} C_DIS
LIN {X 0.010,Y -569.805,Z 1191.265,A 0.000,B 0.000,C 90.000,E1 83.742} C_DIS
LIN {X -0.259,Y -570.980,Z 1191.256,A 0.000,B 0.000,C 90.000,E1 82.129} C_DIS
LIN {X 0.027,Y -571.871,Z 1191.249,A 0.000,B 0.000,C 90.000,E1 80.735} C_DIS
LIN {X -0.231,Y -572.652,Z 1191.241,A 0.000,B 0.000,C 90.000,E1 79.398} C_DIS
LIN {X -0.001,Y -573.331,Z 1191.235,A 0.000,B 0.000,C 90.000,E1 78.285} C_DIS
LIN {X 0.079,Y -574.181,Z 1191.226,A 0.000,B 0.000,C 90.000,E1 76.645} C_DIS
LIN {X -0.051,Y -575.157,Z 1191.215,A 0.000,B 0.000,C 90.000,E1 74.755} C_DIS
LIN {X -0.201,Y -576.251,Z 1191.203,A 0.000,B 0.000,C 90.000,E1 72.598} C_DIS
LIN {X -0.154,Y -577.186,Z 1191.194,A 0.000,B 0.000,C 90.000,E1 70.967} C_DIS
LIN {X -0.255,Y -578.534,Z 1191.184,A 0.000,B 0.000,C 90.000,E1 69.082} C_DIS
LIN {X 0.119,Y -580.684,Z 1191.170,A 0.000,B 0.000,C 90.000,E1 66.613} C_DIS
LIN {X -0.037,Y -581.962,Z 1191.163,A 0.000,B 0.000,C 90.000,E1 65.281} C_DIS
LIN {X 0.104,Y -583.758,Z 1191.152,A 0.000,B 0.000,C 90.000,E1 63.384} C_DIS
LIN {X 0.267,Y -585.142,Z 1191.145,A 0.000,B 0.000,C 90.000,E1 62.025} C_DIS
LIN {X -0.182,Y -586.664,Z 1191.136,A 0.000,B 0.000,C 90.000,E1 60.461} C_DIS
LIN {X -0.194,Y -587.835,Z 1191.128,A 0.000,B 0.000,C 90.000,E1 59.125} C_DIS
LIN {X -0.185,Y -588.929,Z 1191.121,A 0.000,B 0.000,C 90.000,E1 57.788} C_DIS
LIN {X 0.156,Y -589.963,Z 1191.114,A 0.000,B 0.000,C 90.000,E1 56.421} C_DIS
LIN {X -0.109,Y -591.164,Z 1191.105,A 0.000,B 0.000,C 90.000,E1 54.848} C_DIS
LIN {X -0.148,Y -592.296,Z 1191.096,A 0.000,B 0.000,C 90.000,E1 53.256} C_DIS
LIN {X 0.069,Y -593.514,Z 1191.085,A 0.000,B 0.000,C 90.000,E1 51.376} C_DIS
LIN {X -0.356,Y -594.095,Z 1191.080,A 0.000,B 0.000,C 90.000,E1 50.356} C_DIS
LIN {X -0.179,Y -594.825,Z 1191.072,A 0.000,B 0.000,C 90.000,E1 49.013} C_DIS
LIN {X 0.167,Y -595.269,Z 1191.063,A 0.000,B 0.000,C 90.000,E1 47.391} C_DIS
LIN {X -0.303,Y -595.426,Z 1191.057,A 0.000,B 0.000,C 90.000,E1 46.377} C_DIS
LIN {X 0.260,Y -595.404,Z 1191.050,A 0.000,B 0.000,C 90.000,E1 45.000} C_DIS
LIN {X 0.002,Y -595.275,Z 1191.046,A 0.000,B 0.000,C 90.000,E1 44.231} C_DIS
LIN {X -0.248,Y -595.018,Z 1191.041,A 0.000,B 0.000,C 90.000,E1 43.461} C_DIS
LIN {X 0.346,Y -594.611,Z 1191.037,A 0.000,B 0.000,C 90.000,E1 42.609} C_DIS
LIN {X -0.135,Y -593.973,Z 1191.031,A 0.000,B 0.000,C 90.000,E1 41.595} C_DIS
LIN {X -0.207,Y -592.750,Z 1191.022,A 0.000,B 0.000,C 90.000,E1 40.011} C_DIS
LIN {X 0.187,Y -591.761,Z 1191.016,A 0.000,B 0.000,C 90.000,E1 38.910} C_DIS
LIN {X 0.359,Y -590.855,Z 1191.012,A 0.000,B 0.000,C 90.000,E1 38.096} C_DIS
LIN {X -0.105,Y -589.472,Z 1191.006,A 0.000,B 0.000,C 90.000,E1 37.076} C_DIS
LIN {X 0.079,Y -587.468,Z 1190.999,A 0.000,B 0.000,C 90.000,E1 35.724} C_DIS
LIN {X -0.112,Y -584.773,Z 1190.991,A 0.000,B 0.000,C 90.000,E1 34.405} C_DIS
LIN {X -0.071,Y -583.504,Z 1190.988,A 0.000,B 0.000,C 90.000,E1 33.865} C_DIS
LIN {X 0.138,Y -581.251,Z 1190.984,A 0.000,B 0.000,C 90.000,E1 33.038} C_DIS
LIN {X -0.170,Y -578.728,Z 1190.979,A 0.000,B 0.000,C 90.000,E1 32.260} C_DIS
LIN {X -0.171,Y -576.859,Z 1190.976,A 0.000,B 0.000,C 90.000,E1 31.720} C_DIS
LIN {X 0.280,Y -572.558,Z 1190.970,A 0.000,B 0.000,C 90.000,E1 30.590} C_DIS
LIN {X 0.145,Y -569.407,Z 1190.966,A 0.000,B 0.000,C 90.000,E1 29.922} C_DIS
LIN {X -0.295,Y -565.989,Z 1190.963,A 0.000,B 0.000,C 90.000,E1 29.283} C_DIS
LIN {X 0.104,Y -563.026,Z 1190.959,A 0.000,B 0.000,C 90.000,E1 28.693} C_DIS
LIN {X -0.118,Y -559.122,Z 1190.956,A 0.000,B 0.000,C 90.000,E1 28.025} C_DIS
LIN {X -0.034,Y -555.751,Z 1190.953,A 0.000,B 0.000,C 90.000,E1 27.462} C_DIS
LIN {X 0.057,Y -550.412,Z 1190.948,A 0.000,B 0.000,C 90.000,E1 26.616} C_DIS
LIN {X 0.085,Y -546.526,Z 1190.945,A 0.000,B 0.000,C 90.000,E1 26.052} C_DIS
LIN {X 0.279,Y -541.193,Z 1190.941,A 0.000,B 0.000,C 90.000,E1 25.335} C_DIS
LIN {X -0.019,Y -534.338,Z 1190.936,A 0.000,B 0.000,C 90.000,E1 24.515} C_DIS
LIN {X 0.234,Y -528.167,Z 1190.932,A 0.000,B 0.000,C 90.000,E1 23.770} C_DIS
LIN {X -0.068,Y -520.418,Z 1190.927,A 0.000,B 0.000,C 90.000,E1 22.950} C_DIS
LIN {X -0.025,Y -513.886,Z 1190.924,A 0.000,B 0.000,C 90.000,E1 22.259} C_DIS
LIN {X 0.113,Y -504.359,Z 1190.918,A 0.000,B 0.000,C 90.000,E1 21.280} C_DIS
LIN {X -0.141,Y -493.183,Z 1190.912,A 0.000,B 0.000,C 90.000,E1 20.248} C_DIS
LIN {X -0.008,Y -484.573,Z 1190.908,A 0.000,B 0.000,C 90.000,E1 19.450} C_DIS
LIN {X 0.076,Y -474.624,Z 1190.903,A 0.000,B 0.000,C 90.000,E1 18.544} C_DIS
LIN {X -0.201,Y -468.805,Z 1190.900,A 0.000,B 0.000,C 90.000,E1 18.055} C_DIS
LIN {X 0.201,Y -451.392,Z 1190.891,A 0.000,B 0.000,C 90.000,E1 16.441} C_DIS
LIN {X 0.004,Y -429.741,Z 1190.880,A 0.000,B 0.000,C 90.000,E1 14.356} C_DIS
LIN {X 0.082,Y -414.275,Z 1190.870,A 0.000,B 0.000,C 90.000,E1 12.647} C_DIS
LIN {X -0.110,Y -403.533,Z 1190.863,A 0.000,B 0.000,C 90.000,E1 11.366} C_DIS
LIN {X 0.108,Y -398.583,Z 1190.859,A 0.000,B 0.000,C 90.000,E1 10.658} C_DIS
LIN {X -0.053,Y -395.546,Z 1190.857,A 0.000,B 0.000,C 90.000,E1 10.197} C_DIS
LIN {X -0.198,Y -393.907,Z 1190.855,A 0.000,B 0.000,C 90.000,E1 9.849} C_DIS
LIN {X 0.122,Y -393.379,Z 1190.854,A 0.000,B 0.000,C 90.000,E1 9.670} C_DIS
LIN {X 0.083,Y -393.367,Z 1190.854,A 0.000,B 0.000,C 90.000,E1 9.670} C_DIS
LIN {X 0.001,Y -393.244,Z 1190.852,A 0.000,B 0.000,C 90.000,E1 9.378} C_DIS
LIN {X 0.079,Y -394.560,Z 1190.849,A 0.000,B 0.000,C 90.000,E1 8.746} C_DIS
LIN {X 0.148,Y -397.383,Z 1190.845,A 0.000,B 0.000,C 90.000,E1 7.992} C_DIS
LIN {X 0.170,Y -401.288,Z 1190.841,A 0.000,B 0.000,C 90.000,E1 7.352} C_DIS
LIN {X 0.134,Y -402.507,Z 1190.840,A 0.000,B 0.000,C 90.000,E1 7.182} C_DIS
LIN {X 0.087,Y -405.666,Z 1190.838,A 0.000,B 0.000,C 90.000,E1 6.834} C_DIS
LIN {X 0.199,Y -411.152,Z 1190.835,A 0.000,B 0.000,C 90.000,E1 6.315} C_DIS
LIN {X 0.126,Y -428.390,Z 1190.828,A 0.000,B 0.000,C 90.000,E1 4.992} C_DIS
LIN {X -0.092,Y -437.942,Z 1190.824,A 0.000,B 0.000,C 90.000,E1 4.302} C_DIS
LIN {X 0.061,Y -458.871,Z 1190.815,A 0.000,B 0.000,C 90.000,E1 2.751} C_DIS
LIN {X 0.073,Y -466.765,Z 1190.812,A 0.000,B 0.000,C 90.000,E1 2.178} C_DIS
LIN {X -0.129,Y -476.160,Z 1190.808,A 0.000,B 0.000,C 90.000,E1 1.489} C_DIS
LIN {X 0.071,Y -483.784,Z 1190.805,A 0.000,B 0.000,C 90.000,E1 0.859} C_DIS
LIN {X 0.079,Y -491.149,Z 1190.801,A 0.000,B 0.000,C 90.000,E1 0.229} C_DIS
LIN {X 0.038,Y -497.369,Z 1190.798,A 0.000,B 0.000,C 90.000,E1 359.656} C_DIS
LIN {X 0.050,Y -504.119,Z 1190.794,A 0.000,B 0.000,C 90.000,E1 358.969} C_DIS
LIN {X 0.020,Y -511.779,Z 1190.790,A 0.000,B 0.000,C 90.000,E1 358.108} C_DIS
LIN {X -0.146,Y -516.702,Z 1190.786,A 0.000,B 0.000,C 90.000,E1 357.535} C_DIS
LIN {X -0.024,Y -522.307,Z 1190.782,A 0.000,B 0.000,C 90.000,E1 356.788} C_DIS
LIN {X 0.117,Y -527.430,Z 1190.778,A 0.000,B 0.000,C 90.000,E1 356.045} C_DIS
LIN {X 0.089,Y -531.227,Z 1190.775,A 0.000,B 0.000,C 90.000,E1 355.469} C_DIS
LIN {X -0.183,Y -535.469,Z 1190.771,A 0.000,B 0.000,C 90.000,E1 354.780} C_DIS
LIN {X 0.113,Y -539.228,Z 1190.767,A 0.000,B 0.000,C 90.000,E1 354.033} C_DIS
LIN {X -0.033,Y -542.714,Z 1190.763,A 0.000,B 0.000,C 90.000,E1 353.337} C_DIS
LIN {X -0.213,Y -545.811,Z 1190.759,A 0.000,B 0.000,C 90.000,E1 352.648} C_DIS
LIN {X -0.019,Y -549.185,Z 1190.754,A 0.000,B 0.000,C 90.000,E1 351.781} C_DIS
LIN {X 0.209,Y -552.275,Z 1190.750,A 0.000,B 0.000,C 90.000,E1 350.914} C_DIS
LIN {X 0.142,Y -555.869,Z 1190.744,A 0.000,B 0.000,C 90.000,E1 349.803} C_DIS
LIN {X 0.028,Y -559.061,Z 1190.737,A 0.000,B 0.000,C 90.000,E1 348.701} C_DIS
LIN {X 0.061,Y -561.955,Z 1190.731,A 0.000,B 0.000,C 90.000,E1 347.589} C_DIS
LIN {X 0.265,Y -564.591,Z 1190.725,A 0.000,B 0.000,C 90.000,E1 346.464} C_DIS
LIN {X -0.176,Y -567.097,Z 1190.719,A 0.000,B 0.000,C 90.000,E1 345.408} C_DIS
LIN {X -0.117,Y -570.036,Z 1190.711,A 0.000,B 0.000,C 90.000,E1 344.031} C_DIS
LIN {X -0.183,Y -573.726,Z 1190.701,A 0.000,B 0.000,C 90.000,E1 342.127} C_DIS
LIN {X -0.194,Y -575.638,Z 1190.695,A 0.000,B 0.000,C 90.000,E1 341.040} C_DIS
LIN {X 0.015,Y -577.283,Z 1190.689,A 0.000,B 0.000,C 90.000,E1 339.934} C_DIS
LIN {X 0.048,Y -578.654,Z 1190.683,A 0.000,B 0.000,C 90.000,E1 338.847} C_DIS
LIN {X 0.129,Y -579.508,Z 1190.678,A 0.000,B 0.000,C 90.000,E1 338.028} C_DIS
LIN {X -0.138,Y -580.293,Z 1190.672,A 0.000,B 0.000,C 90.000,E1 336.975} C_DIS
LIN {X -0.259,Y -580.535,Z 1190.668,A 0.000,B 0.000,C 90.000,E1 336.177} C_DIS
LIN {X -0.147,Y -580.401,Z 1190.663,A 0.000,B 0.000,C 90.000,E1 335.357} C_DIS
LIN {X -0.036,Y -579.985,Z 1190.659,A 0.000,B 0.000,C 90.000,E1 334.537} C_DIS
LIN {X 0.069,Y -579.180,Z 1190.654,A 0.000,B 0.000,C 90.000,E1 333.717} C_DIS
LIN {X 0.047,Y -578.450,Z 1190.651,A 0.000,B 0.000,C 90.000,E1 333.179} C_DIS
LIN {X 0.132,Y -576.936,Z 1190.647,A 0.000,B 0.000,C 90.000,E1 332.359} C_DIS
LIN {X -0.042,Y -575.178,Z 1190.642,A 0.000,B 0.000,C 90.000,E1 331.563} C_DIS
LIN {X 0.112,Y -572.294,Z 1190.636,A 0.000,B 0.000,C 90.000,E1 330.461} C_DIS
LIN {X 0.065,Y -570.451,Z 1190.633,A 0.000,B 0.000,C 90.000,E1 329.921} C_DIS
LIN {X -0.105,Y -569.412,Z 1190.631,A 0.000,B 0.000,C 90.000,E1 329.665} C_DIS
LIN {X 0.135,Y -565.750,Z 1190.627,A 0.000,B 0.000,C 90.000,E1 328.820} C_DIS
LIN {X 0.040,Y -562.724,Z 1190.624,A 0.000,B 0.000,C 90.000,E1 328.280} C_DIS
LIN {X 0.117,Y -558.310,Z 1190.620,A 0.000,B 0.000,C 90.000,E1 327.582} C_DIS
LIN {X -0.139,Y -553.426,Z 1190.616,A 0.000,B 0.000,C 90.000,E1 326.914} C_DIS
LIN {X -0.011,Y -549.152,Z 1190.613,A 0.000,B 0.000,C 90.000,E1 326.342} C_DIS
LIN {X -0.215,Y -544.650,Z 1190.610,A 0.000,B 0.000,C 90.000,E1 325.801} C_DIS
LIN {X 0.156,Y -538.735,Z 1190.606,A 0.000,B 0.000,C 90.000,E1 325.055} C_DIS
LIN {X 0.180,Y -531.252,Z 1190.601,A 0.000,B 0.000,C 90.000,E1 324.196} C_DIS
LIN {X 0.251,Y -523.800,Z 1190.597,A 0.000,B 0.000,C 90.000,E1 323.336} C_DIS
LIN {X 0.043,Y -520.340,Z 1190.594,A 0.000,B 0.000,C 90.000,E1 322.924} C_DIS
LIN {X 0.004,Y -517.142,Z 1190.591,A 0.000,B 0.000,C 90.000,E1 322.431} C_DIS
LIN {X -0.003,Y -514.837,Z 1190.589,A 0.000,B 0.000,C 90.000,E1 321.949} C_DIS
LIN {X 0.208,Y -513.301,Z 1190.585,A 0.000,B 0.000,C 90.000,E1 321.331} C_DIS
LIN {X -0.223,Y -512.735,Z 1190.581,A 0.000,B 0.000,C 90.000,E1 320.642} C_DIS
LIN {X -0.303,Y -512.604,Z 1190.580,A 0.000,B 0.000,C 90.000,E1 320.356} C_DIS
LIN {X -0.054,Y -513.296,Z 1190.571,A 0.000,B 0.000,C 90.000,E1 318.852} C_DIS
LIN {X -0.179,Y -514.212,Z 1190.563,A 0.000,B 0.000,C 90.000,E1 317.391} C_DIS
LIN {X -0.204,Y -514.839,Z 1190.557,A 0.000,B 0.000,C 90.000,E1 316.215} C_DIS
LIN {X 0.219,Y -516.040,Z 1190.545,A 0.000,B 0.000,C 90.000,E1 314.109} C_DIS
LIN {X -0.235,Y -516.858,Z 1190.537,A 0.000,B 0.000,C 90.000,E1 312.690} C_DIS
LIN {X -0.022,Y -517.995,Z 1190.527,A 0.000,B 0.000,C 90.000,E1 310.906} C_DIS
LIN {X 0.119,Y -518.542,Z 1190.522,A 0.000,B 0.000,C 90.000,E1 310.011} C_DIS
LIN {X 0.151,Y -519.481,Z 1190.514,A 0.000,B 0.000,C 90.000,E1 308.543} C_DIS
LIN {X 0.199,Y -520.284,Z 1190.506,A 0.000,B 0.000,C 90.000,E1 307.076} C_DIS
LIN {X -0.113,Y -521.209,Z 1190.496,A 0.000,B 0.000,C 90.000,E1 305.358} C_DIS
LIN {X 0.151,Y -522.057,Z 1190.487,A 0.000,B 0.000,C 90.000,E1 303.579} C_DIS
LIN {X 0.051,Y -522.771,Z 1190.479,A 0.000,B 0.000,C 90.000,E1 302.133} C_DIS
LIN {X 0.127,Y -523.383,Z 1190.470,A 0.000,B 0.000,C 90.000,E1 300.669} C_DIS
LIN {X 0.216,Y -523.773,Z 1190.462,A 0.000,B 0.000,C 90.000,E1 299.205} C_DIS
LIN {X 0.051,Y -524.083,Z 1190.454,A 0.000,B 0.000,C 90.000,E1 297.769} C_DIS
LIN {X 0.036,Y -524.315,Z 1190.445,A 0.000,B 0.000,C 90.000,E1 296.027} C_DIS
LIN {X -0.116,Y -524.379,Z 1190.437,A 0.000,B 0.000,C 90.000,E1 294.591} C_DIS
LIN {X 0.116,Y -524.225,Z 1190.427,A 0.000,B 0.000,C 90.000,E1 292.823} C_DIS
LIN {X -0.069,Y -524.155,Z 1190.417,A 0.000,B 0.000,C 90.000,E1 291.099} C_DIS
LIN {X 0.232,Y -523.976,Z 1190.408,A 0.000,B 0.000,C 90.000,E1 289.322} C_DIS
LIN {X -0.123,Y -523.775,Z 1190.403,A 0.000,B 0.000,C 90.000,E1 288.489} C_DIS
LIN {X -0.162,Y -523.208,Z 1190.395,A 0.000,B 0.000,C 90.000,E1 287.040} C_DIS
LIN {X 0.135,Y -522.599,Z 1190.388,A 0.000,B 0.000,C 90.000,E1 285.843} C_DIS
LIN {X -0.090,Y -521.484,Z 1190.378,A 0.000,B 0.000,C 90.000,E1 284.120} C_DIS
LIN {X 0.037,Y -520.027,Z 1190.367,A 0.000,B 0.000,C 90.000,E1 282.063} C_DIS
LIN {X 0.023,Y -518.930,Z 1190.357,A 0.000,B 0.000,C 90.000,E1 280.310} C_DIS
LIN {X -0.108,Y -518.012,Z 1190.348,A 0.000,B 0.000,C 90.000,E1 278.568} C_DIS
LIN {X 0.179,Y -517.119,Z 1190.338,A 0.000,B 0.000,C 90.000,E1 276.777} C_DIS
LIN {X -0.021,Y -516.354,Z 1190.331,A 0.000,B 0.000,C 90.000,E1 275.625} C_DIS
LIN {X 0.208,Y -515.445,Z 1190.323,A 0.000,B 0.000,C 90.000,E1 274.131} C_DIS
LIN {X -0.099,Y -514.628,Z 1190.315,A 0.000,B 0.000,C 90.000,E1 272.694} C_DIS
LIN {X -0.012,Y -513.794,Z 1190.305,A 0.000,B 0.000,C 90.000,E1 270.917} C_DIS
LIN {X 0.126,Y -513.105,Z 1190.297,A 0.000,B 0.000,C 90.000,E1 269.427} C_DIS
LIN {X -0.189,Y -512.515,Z 1190.290,A 0.000,B 0.000,C 90.000,E1 268.282} C_DIS
LIN {X -0.128,Y -511.368,Z 1190.281,A 0.000,B 0.000,C 90.000,E1 266.502} C_DIS
LIN {X 0.004,Y -510.306,Z 1190.272,A 0.000,B 0.000,C 90.000,E1 265.008} C_DIS
LIN {X 0.108,Y -508.865,Z 1190.264,A 0.000,B 0.000,C 90.000,E1 263.514} C_DIS
LIN {X 0.130,Y -507.009,Z 1190.253,A 0.000,B 0.000,C 90.000,E1 261.432} C_DIS
LIN {X 0.181,Y -505.292,Z 1190.241,A 0.000,B 0.000,C 90.000,E1 259.342} C_DIS
LIN {X -0.042,Y -504.314,Z 1190.234,A 0.000,B 0.000,C 90.000,E1 258.173} C_DIS
LIN {X 0.195,Y -502.798,Z 1190.224,A 0.000,B 0.000,C 90.000,E1 256.353} C_DIS
LIN {X -0.044,Y -501.043,Z 1190.213,A 0.000,B 0.000,C 90.000,E1 254.283} C_DIS
LIN {X -0.051,Y -499.483,Z 1190.201,A 0.000,B 0.000,C 90.000,E1 252.181} C_DIS
LIN {X 0.043,Y -498.557,Z 1190.194,A 0.000,B 0.000,C 90.000,E1 250.967} C_DIS
LIN {X 0.068,Y -496.989,Z 1190.184,A 0.000,B 0.000,C 90.000,E1 249.156} C_DIS
LIN {X -0.061,Y -495.319,Z 1190.174,A 0.000,B 0.000,C 90.000,E1 247.358} C_DIS
LIN {X -0.069,Y -493.820,Z 1190.166,A 0.000,B 0.000,C 90.000,E1 245.845} C_DIS
LIN {X 0.096,Y -492.568,Z 1190.159,A 0.000,B 0.000,C 90.000,E1 244.613} C_DIS
LIN {X -0.198,Y -490.811,Z 1190.151,A 0.000,B 0.000,C 90.000,E1 243.127} C_DIS
LIN {X -0.097,Y -489.311,Z 1190.144,A 0.000,B 0.000,C 90.000,E1 241.897} C_DIS
LIN {X 0.217,Y -487.355,Z 1190.135,A 0.000,B 0.000,C 90.000,E1 240.333} C_DIS
LIN {X -0.123,Y -484.996,Z 1190.125,A 0.000,B 0.000,C 90.000,E1 238.535} C_DIS
LIN {X -0.261,Y -482.555,Z 1190.115,A 0.000,B 0.000,C 90.000,E1 236.707} C_DIS
LIN {X -0.110,Y -479.696,Z 1190.103,A 0.000,B 0.000,C 90.000,E1 234.529} C_DIS
LIN {X -0.019,Y -477.742,Z 1190.094,A 0.000,B 0.000,C 90.000,E1 232.970} C_DIS
LIN {X -0.094,Y -474.983,Z 1190.082,A 0.000,B 0.000,C 90.000,E1 230.803} C_DIS
LIN {X 0.118,Y -473.099,Z 1190.074,A 0.000,B 0.000,C 90.000,E1 229.218} C_DIS
LIN {X -0.059,Y -471.080,Z 1190.065,A 0.000,B 0.000,C 90.000,E1 227.676} C_DIS
LIN {X 0.112,Y -467.244,Z 1190.047,A 0.000,B 0.000,C 90.000,E1 224.514} C_DIS
LIN {X 0.078,Y -464.597,Z 1190.032,A 0.000,B 0.000,C 90.000,E1 221.676} C_DIS
LIN {X 0.199,Y -463.445,Z 1190.012,A 0.000,B 0.000,C 90.000,E1 218.177} C_DIS
LIN {X 0.108,Y -463.469,Z 1190.007,A 0.000,B 0.000,C 90.000,E1 217.237} C_DIS
LIN {X -0.105,Y -463.437,Z 1189.998,A 0.000,B 0.000,C 90.000,E1 215.678} C_DIS
LIN {X -0.187,Y -463.654,Z 1189.988,A 0.000,B 0.000,C 90.000,E1 213.785} C_DIS
LIN {X 0.186,Y -465.882,Z 1189.968,A 0.000,B 0.000,C 90.000,E1 210.256} C_DIS
LIN {X -0.185,Y -468.672,Z 1189.953,A 0.000,B 0.000,C 90.000,E1 207.462} C_DIS
LIN {X -0.217,Y -473.696,Z 1189.930,A 0.000,B 0.000,C 90.000,E1 203.387} C_DIS
LIN {X -0.050,Y -481.072,Z 1189.907,A 0.000,B 0.000,C 90.000,E1 199.322} C_DIS
LIN {X 0.174,Y -490.292,Z 1189.887,A 0.000,B 0.000,C 90.000,E1 195.607} C_DIS
LIN {X 0.189,Y -497.467,Z 1189.873,A 0.000,B 0.000,C 90.000,E1 193.175} C_DIS
LIN {X 0.147,Y -504.095,Z 1189.862,A 0.000,B 0.000,C 90.000,E1 191.074} C_DIS
LIN {X 0.166,Y -511.997,Z 1189.848,A 0.000,B 0.000,C 90.000,E1 188.690} C_DIS
LIN {X -0.058,Y -516.948,Z 1189.840,A 0.000,B 0.000,C 90.000,E1 187.239} C_DIS
LIN {X -0.254,Y -520.873,Z 1189.834,A 0.000,B 0.000,C 90.000,E1 186.087} C_DIS
LIN {X 0.082,Y -527.687,Z 1189.822,A 0.000,B 0.000,C 90.000,E1 184.012} C_DIS
LIN {X -0.009,Y -530.586,Z 1189.818,A 0.000,B 0.000,C 90.000,E1 183.154} C_DIS
LIN {X -0.034,Y -536.398,Z 1189.808,A 0.000,B 0.000,C 90.000,E1 181.432} C_DIS
LIN {X 0.083,Y -544.051,Z 1189.795,A 0.000,B 0.000,C 90.000,E1 179.141} C_DIS
LIN {X -0.218,Y -549.781,Z 1189.786,A 0.000,B 0.000,C 90.000,E1 177.478} C_DIS
LIN {X 0.082,Y -554.419,Z 1189.778,A 0.000,B 0.000,C 90.000,E1 176.045} C_DIS
LIN {X -0.123,Y -558.130,Z 1189.772,A 0.000,B 0.000,C 90.000,E1 174.951} C_DIS
LIN {X -0.047,Y -563.533,Z 1189.763,A 0.000,B 0.000,C 90.000,E1 173.280} C_DIS
LIN {X 0.214,Y -568.880,Z 1189.754,A 0.000,B 0.000,C 90.000,E1 171.602} C_DIS
LIN {X -0.173,Y -573.266,Z 1189.746,A 0.000,B 0.000,C 90.000,E1 170.274} C_DIS
LIN {X 0.064,Y -576.741,Z 1189.740,A 0.000,B 0.000,C 90.000,E1 169.162} C_DIS
LIN {X -0.093,Y -582.783,Z 1189.729,A 0.000,B 0.000,C 90.000,E1 167.285} C_DIS
LIN {X -0.038,Y -587.093,Z 1189.722,A 0.000,B 0.000,C 90.000,E1 165.936} C_DIS
LIN {X 0.232,Y -591.358,Z 1189.714,A 0.000,B 0.000,C 90.000,E1 164.574} C_DIS
LIN {X -0.130,Y -596.455,Z 1189.706,A 0.000,B 0.000,C 90.000,E1 163.015} C_DIS
LIN {X -0.098,Y -600.705,Z 1189.698,A 0.000,B 0.000,C 90.000,E1 161.692} C_DIS
LIN {X 0.284,Y -604.023,Z 1189.693,A 0.000,B 0.000,C 90.000,E1 160.604} C_DIS
LIN {X -0.141,Y -608.113,Z 1189.685,A 0.000,B 0.000,C 90.000,E1 159.337} C_DIS
LIN {X -0.020,Y -611.312,Z 1189.679,A 0.000,B 0.000,C 90.000,E1 158.284} C_DIS
LIN {X 0.119,Y -615.346,Z 1189.672,A 0.000,B 0.000,C 90.000,E1 156.975} C_DIS
LIN {X 0.061,Y -620.053,Z 1189.664,A 0.000,B 0.000,C 90.000,E1 155.433} C_DIS
LIN {X 0.042,Y -624.561,Z 1189.655,A 0.000,B 0.000,C 90.000,E1 153.896} C_DIS
LIN {X 0.102,Y -628.132,Z 1189.648,A 0.000,B 0.000,C 90.000,E1 152.615} C_DIS
LIN {X 0.189,Y -630.952,Z 1189.642,A 0.000,B 0.000,C 90.000,E1 151.591} C_DIS
LIN {X 0.130,Y -634.984,Z 1189.634,A 0.000,B 0.000,C 90.000,E1 150.078} C_DIS
LIN {X 0.060,Y -637.559,Z 1189.628,A 0.000,B 0.000,C 90.000,E1 149.076} C_DIS
LIN {X 0.409,Y -640.565,Z 1189.621,A 0.000,B 0.000,C 90.000,E1 147.788} C_DIS
LIN {X -0.078,Y -643.409,Z 1189.614,A 0.000,B 0.000,C 90.000,E1 146.580} C_DIS
LIN {X 0.255,Y -645.000,Z 1189.610,A 0.000,B 0.000,C 90.000,E1 145.801} C_DIS
LIN {X 0.187,Y -647.533,Z 1189.603,A 0.000,B 0.000,C 90.000,E1 144.562} C_DIS
LIN {X 0.008,Y -649.845,Z 1189.596,A 0.000,B 0.000,C 90.000,E1 143.336} C_DIS
LIN {X -0.126,Y -652.146,Z 1189.589,A 0.000,B 0.000,C 90.000,E1 142.110} C_DIS
LIN {X -0.343,Y -656.365,Z 1189.577,A 0.000,B 0.000,C 90.000,E1 139.908} C_DIS
LIN {X -0.433,Y -658.357,Z 1189.572,A 0.000,B 0.000,C 90.000,E1 138.933} C_DIS
LIN {X 0.385,Y -661.549,Z 1189.563,A 0.000,B 0.000,C 90.000,E1 137.391} C_DIS
LIN {X -0.154,Y -664.636,Z 1189.555,A 0.000,B 0.000,C 90.000,E1 135.972} C_DIS
LIN {X -0.159,Y -669.483,Z 1189.543,A 0.000,B 0.000,C 90.000,E1 133.785} C_DIS
LIN {X -0.020,Y -674.093,Z 1189.532,A 0.000,B 0.000,C 90.000,E1 131.838} C_DIS
LIN {X 0.172,Y -677.542,Z 1189.524,A 0.000,B 0.000,C 90.000,E1 130.378} C_DIS
LIN {X -0.043,Y -680.551,Z 1189.518,A 0.000,B 0.000,C 90.000,E1 129.197} C_DIS
LIN {X -0.026,Y -684.673,Z 1189.509,A 0.000,B 0.000,C 90.000,E1 127.523} C_DIS
LIN {X 0.415,Y -687.664,Z 1189.502,A 0.000,B 0.000,C 90.000,E1 126.297} C_DIS
LIN {X -0.100,Y -690.055,Z 1189.497,A 0.000,B 0.000,C 90.000,E1 125.391} C_DIS
LIN {X 0.271,Y -693.867,Z 1189.487,A 0.000,B 0.000,C 90.000,E1 123.706} C_DIS
LIN {X -0.205,Y -695.475,Z 1189.484,A 0.000,B 0.000,C 90.000,E1 123.038} C_DIS
LIN {X -0.387,Y -697.996,Z 1189.477,A 0.000,B 0.000,C 90.000,E1 121.878} C_DIS
LIN {X -0.278,Y -700.774,Z 1189.469,A 0.000,B 0.000,C 90.000,E1 120.463} C_DIS
LIN {X -0.141,Y -702.814,Z 1189.463,A 0.000,B 0.000,C 90.000,E1 119.283} C_DIS
LIN {X 0.031,Y -704.663,Z 1189.456,A 0.000,B 0.000,C 90.000,E1 118.103} C_DIS
LIN {X 0.269,Y -705.591,Z 1189.452,A 0.000,B 0.000,C 90.000,E1 117.385} C_DIS
LIN {X 0.194,Y -706.184,Z 1189.448,A 0.000,B 0.000,C 90.000,E1 116.693} C_DIS
LIN {X -0.206,Y -706.664,Z 1189.443,A 0.000,B 0.000,C 90.000,E1 115.796} C_DIS
LIN {X 0.040,Y -706.712,Z 1189.439,A 0.000,B 0.000,C 90.000,E1 115.079} C_DIS
LIN {X -0.312,Y -706.447,Z 1189.437,A 0.000,B 0.000,C 90.000,E1 114.643} C_DIS
LIN {X -0.018,Y -705.683,Z 1189.434,A 0.000,B 0.000,C 90.000,E1 114.155} C_DIS
LIN {X 0.273,Y -705.222,Z 1189.433,A 0.000,B 0.000,C 90.000,E1 113.898} C_DIS
LIN {X 0.059,Y -702.567,Z 1189.430,A 0.000,B 0.000,C 90.000,E1 113.334} C_DIS
LIN {X 0.201,Y -701.826,Z 1189.429,A 0.000,B 0.000,C 90.000,E1 113.206} C_DIS
LIN {X 0.337,Y -700.721,Z 1189.428,A 0.000,B 0.000,C 90.000,E1 113.078} C_DIS
LIN {X -0.121,Y -695.837,Z 1189.426,A 0.000,B 0.000,C 90.000,E1 112.695} C_DIS
LIN {X -0.167,Y -694.061,Z 1189.425,A 0.000,B 0.000,C 90.000,E1 112.589} C_DIS
LIN {X 0.276,Y -691.500,Z 1189.425,A 0.000,B 0.000,C 90.000,E1 112.461} C_DIS
LIN {X 0.073,Y -686.809,Z 1189.424,A 0.000,B 0.000,C 90.000,E1 112.333} C_DIS
LIN {X 0.068,Y -683.974,Z 1189.424,A 0.000,B 0.000,C 90.000,E1 112.280} C_DIS
LIN {X -0.231,Y -677.646,Z 1189.424,A 0.000,B 0.000,C 90.000,E1 112.280} C_DIS
LIN {X -0.027,Y -606.814,Z 1189.424,A 0.000,B 0.000,C 90.000,E1 112.259} C_DIS
LIN {X 0.235,Y -601.736,Z 1189.422,A 0.000,B 0.000,C 90.000,E1 111.897} C_DIS
LIN {X -0.258,Y -590.693,Z 1189.417,A 0.000,B 0.000,C 90.000,E1 111.046} C_DIS
LIN {X -0.093,Y -580.602,Z 1189.412,A 0.000,B 0.000,C 90.000,E1 110.248} C_DIS
LIN {X 0.027,Y -571.834,Z 1189.409,A 0.000,B 0.000,C 90.000,E1 109.577} C_DIS
LIN {X 0.188,Y -563.023,Z 1189.405,A 0.000,B 0.000,C 90.000,E1 108.906} C_DIS
LIN {X 0.341,Y -561.943,Z 1189.405,A 0.000,B 0.000,C 90.000,E1 108.779} C_DIS
LIN {X 0.193,Y -559.691,Z 1189.403,A 0.000,B 0.000,C 90.000,E1 108.598} C_DIS
LIN {X 0.153,Y -559.649,Z 1189.403,A 0.000,B 0.000,C 90.000,E1 108.598} C_DIS
LIN {X -0.083,Y -558.799,Z 1189.402,A 0.000,B 0.000,C 90.000,E1 108.417} C_DIS
LIN {X 0.143,Y -557.459,Z 1189.401,A 0.000,B 0.000,C 90.000,E1 108.181} C_DIS
LIN {X 0.101,Y -557.446,Z 1189.401,A 0.000,B 0.000,C 90.000,E1 108.181} C_DIS
LIN {X -0.194,Y -557.906,Z 1189.397,A 0.000,B 0.000,C 90.000,E1 107.457} C_DIS
LIN {X 0.107,Y -559.711,Z 1189.391,A 0.000,B 0.000,C 90.000,E1 106.315} C_DIS
LIN {X -0.158,Y -560.351,Z 1189.388,A 0.000,B 0.000,C 90.000,E1 105.788} C_DIS
LIN {X 0.276,Y -560.525,Z 1189.385,A 0.000,B 0.000,C 90.000,E1 105.190} C_DIS
LIN {X -0.121,Y -560.447,Z 1189.383,A 0.000,B 0.000,C 90.000,E1 104.954} C_DIS
LIN {X 0.312,Y -559.871,Z 1189.380,A 0.000,B 0.000,C 90.000,E1 104.356} C_DIS
LIN {X -0.086,Y -559.008,Z 1189.378,A 0.000,B 0.000,C 90.000,E1 104.120} C_DIS
LIN {X 0.058,Y -558.582,Z 1189.377,A 0.000,B 0.000,C 90.000,E1 103.828} C_DIS
LIN {X -0.170,Y -556.857,Z 1189.373,A 0.000,B 0.000,C 90.000,E1 103.175} C_DIS
LIN {X -0.212,Y -556.848,Z 1189.373,A 0.000,B 0.000,C 90.000,E1 103.175} C_DIS
LIN {X 0.075,Y -556.267,Z 1189.371,A 0.000,B 0.000,C 90.000,E1 102.715} C_DIS
LIN {X -0.211,Y -556.345,Z 1189.369,A 0.000,B 0.000,C 90.000,E1 102.467} C_DIS
LIN {X -0.072,Y -556.181,Z 1189.368,A 0.000,B 0.000,C 90.000,E1 102.187} C_DIS
LIN {X 0.179,Y -556.237,Z 1189.366,A 0.000,B 0.000,C 90.000,E1 101.883} C_DIS
LIN {X 0.005,Y -556.783,Z 1189.362,A 0.000,B 0.000,C 90.000,E1 101.074} C_DIS
LIN {X 0.142,Y -556.822,Z 1189.360,A 0.000,B 0.000,C 90.000,E1 100.782} C_DIS
LIN {X 0.052,Y -558.662,Z 1189.348,A 0.000,B 0.000,C 90.000,E1 98.568} C_DIS
LIN {X 0.182,Y -560.226,Z 1189.338,A 0.000,B 0.000,C 90.000,E1 96.891} C_DIS
LIN {X 0.140,Y -561.307,Z 1189.331,A 0.000,B 0.000,C 90.000,E1 95.511} C_DIS
LIN {X 0.031,Y -562.024,Z 1189.325,A 0.000,B 0.000,C 90.000,E1 94.416} C_DIS
LIN {X 0.018,Y -562.988,Z 1189.317,A 0.000,B 0.000,C 90.000,E1 93.037} C_DIS
LIN {X -0.015,Y -563.967,Z 1189.309,A 0.000,B 0.000,C 90.000,E1 91.661} C_DIS
LIN {X 0.070,Y -565.232,Z 1189.300,A 0.000,B 0.000,C 90.000,E1 90.000} C_DIS
LIN {X -0.136,Y -566.762,Z 1189.288,A 0.000,B 0.000,C 90.000,E1 87.822} C_DIS
LIN {X -0.210,Y -567.557,Z 1189.282,A 0.000,B 0.000,C 90.000,E1 86.731} C_DIS
LIN {X 0.000,Y -568.733,Z 1189.273,A 0.000,B 0.000,C 90.000,E1 85.065} C_DIS
LIN {X 0.112,Y -569.731,Z 1189.265,A 0.000,B 0.000,C 90.000,E1 83.685} C_DIS
LIN {X -0.083,Y -570.887,Z 1189.256,A 0.000,B 0.000,C 90.000,E1 82.064} C_DIS
LIN {X -0.068,Y -571.623,Z 1189.250,A 0.000,B 0.000,C 90.000,E1 80.971} C_DIS
LIN {X -0.140,Y -572.539,Z 1189.241,A 0.000,B 0.000,C 90.000,E1 79.342} C_DIS
LIN {X 0.085,Y -573.203,Z 1189.235,A 0.000,B 0.000,C 90.000,E1 78.229} C_DIS
LIN {X 0.159,Y -574.054,Z 1189.226,A 0.000,B 0.000,C 90.000,E1 76.589} C_DIS
LIN {X 0.022,Y -575.037,Z 1189.215,A 0.000,B 0.000,C 90.000,E1 74.700} C_DIS
LIN {X 0.229,Y -576.287,Z 1189.202,A 0.000,B 0.000,C 90.000,E1 72.236} C_DIS
LIN {X -0.082,Y -577.422,Z 1189.191,A 0.000,B 0.000,C 90.000,E1 70.369} C_DIS
LIN {X -0.209,Y -578.404,Z 1189.183,A 0.000,B 0.000,C 90.000,E1 69.028} C_DIS
LIN {X 0.152,Y -580.620,Z 1189.170,A 0.000,B 0.000,C 90.000,E1 66.561} C_DIS
LIN {X -0.010,Y -581.875,Z 1189.162,A 0.000,B 0.000,C 90.000,E1 65.229} C_DIS
LIN {X -0.272,Y -583.415,Z 1189.153,A 0.000,B 0.000,C 90.000,E1 63.640} C_DIS
LIN {X -0.240,Y -585.057,Z 1189.145,A 0.000,B 0.000,C 90.000,E1 62.025} C_DIS
LIN {X -0.059,Y -586.330,Z 1189.137,A 0.000,B 0.000,C 90.000,E1 60.667} C_DIS
LIN {X -0.081,Y -587.512,Z 1189.130,A 0.000,B 0.000,C 90.000,E1 59.331} C_DIS
LIN {X -0.079,Y -588.620,Z 1189.122,A 0.000,B 0.000,C 90.000,E1 57.995} C_DIS
LIN {X 0.255,Y -589.653,Z 1189.115,A 0.000,B 0.000,C 90.000,E1 56.628} C_DIS
LIN {X 0.192,Y -591.040,Z 1189.104,A 0.000,B 0.000,C 90.000,E1 54.769} C_DIS
LIN {X -0.200,Y -592.141,Z 1189.096,A 0.000,B 0.000,C 90.000,E1 53.210} C_DIS
LIN {X -0.245,Y -593.518,Z 1189.084,A 0.000,B 0.000,C 90.000,E1 51.090} C_DIS
LIN {X -0.094,Y -594.492,Z 1189.073,A 0.000,B 0.000,C 90.000,E1 49.218} C_DIS
LIN {X -0.128,Y -594.853,Z 1189.068,A 0.000,B 0.000,C 90.000,E1 48.162} C_DIS
LIN {X 0.239,Y -595.151,Z 1189.062,A 0.000,B 0.000,C 90.000,E1 47.067} C_DIS
LIN {X -0.031,Y -595.175,Z 1189.054,A 0.000,B 0.000,C 90.000,E1 45.769} C_DIS
LIN {X 0.102,Y -595.105,Z 1189.047,A 0.000,B 0.000,C 90.000,E1 44.433} C_DIS
LIN {X 0.039,Y -594.750,Z 1189.041,A 0.000,B 0.000,C 90.000,E1 43.380} C_DIS
LIN {X -0.210,Y -594.310,Z 1189.037,A 0.000,B 0.000,C 90.000,E1 42.609} C_DIS
LIN {X -0.092,Y -593.476,Z 1189.029,A 0.000,B 0.000,C 90.000,E1 41.272} C_DIS
LIN {X 0.062,Y -592.442,Z 1189.022,A 0.000,B 0.000,C 90.000,E1 39.930} C_DIS
LIN {X -0.011,Y -591.411,Z 1189.016,A 0.000,B 0.000,C 90.000,E1 38.874} C_DIS
LIN {X -0.004,Y -590.177,Z 1189.010,A 0.000,B 0.000,C 90.000,E1 37.810} C_DIS
LIN {X 0.197,Y -588.265,Z 1189.003,A 0.000,B 0.000,C 90.000,E1 36.457} C_DIS
LIN {X -0.024,Y -587.025,Z 1188.998,A 0.000,B 0.000,C 90.000,E1 35.678} C_DIS
LIN {X 0.115,Y -584.235,Z 1188.991,A 0.000,B 0.000,C 90.000,E1 34.326} C_DIS
LIN {X 0.149,Y -582.967,Z 1188.988,A 0.000,B 0.000,C 90.000,E1 33.785} C_DIS
LIN {X -0.287,Y -579.815,Z 1188.982,A 0.000,B 0.000,C 90.000,E1 32.752} C_DIS
LIN {X -0.277,Y -578.070,Z 1188.979,A 0.000,B 0.000,C 90.000,E1 32.212} C_DIS
LIN {X -0.277,Y -576.156,Z 1188.976,A 0.000,B 0.000,C 90.000,E1 31.671} C_DIS
LIN {X 0.334,Y -572.920,Z 1188.971,A 0.000,B 0.000,C 90.000,E1 30.797} C_DIS
LIN {X 0.206,Y -569.927,Z 1188.968,A 0.000,B 0.000,C 90.000,E1 30.129} C_DIS
LIN {X -0.043,Y -565.875,Z 1188.963,A 0.000,B 0.000,C 90.000,E1 29.333} C_DIS
LIN {X 0.079,Y -562.932,Z 1188.960,A 0.000,B 0.000,C 90.000,E1 28.771} C_DIS
LIN {X -0.340,Y -557.393,Z 1188.955,A 0.000,B 0.000,C 90.000,E1 27.847} C_DIS
LIN {X -0.228,Y -552.137,Z 1188.950,A 0.000,B 0.000,C 90.000,E1 27.001} C_DIS
LIN {X 0.056,Y -548.418,Z 1188.947,A 0.000,B 0.000,C 90.000,E1 26.411} C_DIS
LIN {X 0.190,Y -545.436,Z 1188.944,A 0.000,B 0.000,C 90.000,E1 25.976} C_DIS
LIN {X 0.055,Y -539.953,Z 1188.941,A 0.000,B 0.000,C 90.000,E1 25.283} C_DIS
LIN {X -0.100,Y -534.260,Z 1188.937,A 0.000,B 0.000,C 90.000,E1 24.591} C_DIS
LIN {X -0.111,Y -528.099,Z 1188.933,A 0.000,B 0.000,C 90.000,E1 23.875} C_DIS
LIN {X 0.095,Y -521.797,Z 1188.929,A 0.000,B 0.000,C 90.000,E1 23.153} C_DIS
LIN {X -0.002,Y -515.207,Z 1188.925,A 0.000,B 0.000,C 90.000,E1 22.461} C_DIS
LIN {X 0.025,Y -504.315,Z 1188.919,A 0.000,B 0.000,C 90.000,E1 21.354} C_DIS
LIN {X 0.194,Y -492.866,Z 1188.913,A 0.000,B 0.000,C 90.000,E1 20.248} C_DIS
LIN {X 0.157,Y -482.675,Z 1188.907,A 0.000,B 0.000,C 90.000,E1 19.322} C_DIS
LIN {X -0.042,Y -470.929,Z 1188.902,A 0.000,B 0.000,C 90.000,E1 18.290} C_DIS
LIN {X -0.015,Y -454.936,Z 1188.894,A 0.000,B 0.000,C 90.000,E1 16.858} C_DIS
LIN {X -0.139,Y -431.761,Z 1188.881,A 0.000,B 0.000,C 90.000,E1 14.647} C_DIS
LIN {X -0.169,Y -414.976,Z 1188.871,A 0.000,B 0.000,C 90.000,E1 12.827} C_DIS
LIN {X 0.084,Y -402.785,Z 1188.863,A 0.000,B 0.000,C 90.000,E1 11.299} C_DIS
LIN {X 0.094,Y -397.855,Z 1188.859,A 0.000,B 0.000,C 90.000,E1 10.602} C_DIS
LIN {X 0.076,Y -395.693,Z 1188.857,A 0.000,B 0.000,C 90.000,E1 10.254} C_DIS
LIN {X 0.099,Y -394.785,Z 1188.856,A 0.000,B 0.000,C 90.000,E1 10.074} C_DIS
LIN {X 0.100,Y -393.388,Z 1188.854,A 0.000,B 0.000,C 90.000,E1 9.726} C_DIS
LIN {X 0.062,Y -393.378,Z 1188.854,A 0.000,B 0.000,C 90.000,E1 9.726} C_DIS
LIN {X -0.097,Y -393.248,Z 1188.852,A 0.000,B 0.000,C 90.000,E1 9.434} C_DIS
LIN {X 0.020,Y -393.709,Z 1188.851,A 0.000,B 0.000,C 90.000,E1 9.151} C_DIS
LIN {X -0.019,Y -394.469,Z 1188.849,A 0.000,B 0.000,C 90.000,E1 8.803} C_DIS
LIN {X 0.084,Y -397.252,Z 1188.845,A 0.000,B 0.000,C 90.000,E1 8.049} C_DIS
LIN {X -0.032,Y -402.482,Z 1188.840,A 0.000,B 0.000,C 90.000,E1 7.182} C_DIS
LIN {X 0.098,Y -406.432,Z 1188.837,A 0.000,B 0.000,C 90.000,E1 6.720} C_DIS
LIN {X 0.131,Y -411.505,Z 1188.835,A 0.000,B 0.000,C 90.000,E1 6.258} C_DIS
LIN {X 0.140,Y -427.144,Z 1188.828,A 0.000,B 0.000,C 90.000,E1 5.049} C_DIS
LIN {X -0.140,Y -438.336,Z 1188.823,A 0.000,B 0.000,C 90.000,E1 4.245} C_DIS
LIN {X 0.074,Y -459.242,Z 1188.815,A 0.000,B 0.000,C 90.000,E1 2.694} C_DIS
LIN {X 0.101,Y -467.098,Z 1188.812,A 0.000,B 0.000,C 90.000,E1 2.121} C_DIS
LIN {X -0.049,Y -476.442,Z 1188.808,A 0.000,B 0.000,C 90.000,E1 1.432} C_DIS
LIN {X 0.180,Y -484.081,Z 1188.805,A 0.000,B 0.000,C 90.000,E1 0.802} C_DIS
LIN {X -0.176,Y -491.322,Z 1188.801,A 0.000,B 0.000,C 90.000,E1 0.229} C_DIS
LIN {X 0.039,Y -497.278,Z 1188.798,A 0.000,B 0.000,C 90.000,E1 359.656} C_DIS
LIN {X 0.140,Y -503.993,Z 1188.794,A 0.000,B 0.000,C 90.000,E1 358.969} C_DIS
LIN {X 0.140,Y -511.710,Z 1188.790,A 0.000,B 0.000,C 90.000,E1 358.108} C_DIS
LIN {X -0.026,Y -516.657,Z 1188.786,A 0.000,B 0.000,C 90.000,E1 357.535} C_DIS
LIN {X 0.185,Y -522.276,Z 1188.782,A 0.000,B 0.000,C 90.000,E1 356.788} C_DIS
LIN {X -0.108,Y -527.348,Z 1188.778,A 0.000,B 0.000,C 90.000,E1 356.102} C_DIS
LIN {X -0.138,Y -531.185,Z 1188.775,A 0.000,B 0.000,C 90.000,E1 355.527} C_DIS
LIN {X 0.121,Y -535.494,Z 1188.771,A 0.000,B 0.000,C 90.000,E1 354.780} C_DIS
LIN {X 0.208,Y -539.969,Z 1188.766,A 0.000,B 0.000,C 90.000,E1 353.913} C_DIS
LIN {X 0.277,Y -542.804,Z 1188.763,A 0.000,B 0.000,C 90.000,E1 353.337} C_DIS
LIN {X 0.100,Y -545.938,Z 1188.759,A 0.000,B 0.000,C 90.000,E1 352.648} C_DIS
LIN {X 0.278,Y -548.285,Z 1188.756,A 0.000,B 0.000,C 90.000,E1 352.064} C_DIS
LIN {X -0.039,Y -551.471,Z 1188.751,A 0.000,B 0.000,C 90.000,E1 351.254} C_DIS
LIN {X 0.218,Y -554.356,Z 1188.747,A 0.000,B 0.000,C 90.000,E1 350.387} C_DIS
LIN {X 0.084,Y -557.765,Z 1188.741,A 0.000,B 0.000,C 90.000,E1 349.285} C_DIS
LIN {X -0.046,Y -560.099,Z 1188.736,A 0.000,B 0.000,C 90.000,E1 348.465} C_DIS
LIN {X 0.004,Y -562.926,Z 1188.730,A 0.000,B 0.000,C 90.000,E1 347.353} C_DIS
LIN {X -0.162,Y -566.177,Z 1188.722,A 0.000,B 0.000,C 90.000,E1 345.992} C_DIS
LIN {X 0.284,Y -569.182,Z 1188.714,A 0.000,B 0.000,C 90.000,E1 344.574} C_DIS
LIN {X 0.046,Y -571.434,Z 1188.708,A 0.000,B 0.000,C 90.000,E1 343.504} C_DIS
LIN {X -0.004,Y -574.589,Z 1188.699,A 0.000,B 0.000,C 90.000,E1 341.873} C_DIS
LIN {X 0.004,Y -576.476,Z 1188.693,A 0.000,B 0.000,C 90.000,E1 340.786} C_DIS
LIN {X 0.032,Y -578.067,Z 1188.687,A 0.000,B 0.000,C 90.000,E1 339.699} C_DIS
LIN {X 0.280,Y -579.421,Z 1188.681,A 0.000,B 0.000,C 90.000,E1 338.592} C_DIS
LIN {X 0.156,Y -580.210,Z 1188.677,A 0.000,B 0.000,C 90.000,E1 337.794} C_DIS
LIN {X -0.108,Y -580.979,Z 1188.671,A 0.000,B 0.000,C 90.000,E1 336.741} C_DIS
LIN {X 0.008,Y -581.123,Z 1188.666,A 0.000,B 0.000,C 90.000,E1 335.921} C_DIS
LIN {X 0.128,Y -580.936,Z 1188.662,A 0.000,B 0.000,C 90.000,E1 335.101} C_DIS
LIN {X -0.143,Y -580.681,Z 1188.659,A 0.000,B 0.000,C 90.000,E1 334.588} C_DIS
LIN {X -0.028,Y -579.907,Z 1188.654,A 0.000,B 0.000,C 90.000,E1 333.768} C_DIS
LIN {X -0.303,Y -579.228,Z 1188.651,A 0.000,B 0.000,C 90.000,E1 333.256} C_DIS
LIN {X -0.088,Y -577.188,Z 1188.645,A 0.000,B 0.000,C 90.000,E1 332.153} C_DIS
LIN {X 0.249,Y -575.351,Z 1188.641,A 0.000,B 0.000,C 90.000,E1 331.307} C_DIS
LIN {X -0.218,Y -573.202,Z 1188.636,A 0.000,B 0.000,C 90.000,E1 330.539} C_DIS
LIN {X 0.354,Y -570.492,Z 1188.632,A 0.000,B 0.000,C 90.000,E1 329.665} C_DIS
LIN {X 0.025,Y -566.265,Z 1188.626,A 0.000,B 0.000,C 90.000,E1 328.742} C_DIS
LIN {X -0.162,Y -562.329,Z 1188.623,A 0.000,B 0.000,C 90.000,E1 328.074} C_DIS
LIN {X -0.084,Y -557.755,Z 1188.619,A 0.000,B 0.000,C 90.000,E1 327.375} C_DIS
LIN {X -0.228,Y -553.808,Z 1188.616,A 0.000,B 0.000,C 90.000,E1 326.834} C_DIS
LIN {X 0.237,Y -548.401,Z 1188.612,A 0.000,B 0.000,C 90.000,E1 326.087} C_DIS
LIN {X 0.022,Y -543.870,Z 1188.609,A 0.000,B 0.000,C 90.000,E1 325.548} C_DIS
LIN {X 0.083,Y -539.069,Z 1188.605,A 0.000,B 0.000,C 90.000,E1 324.975} C_DIS
LIN {X 0.118,Y -531.537,Z 1188.601,A 0.000,B 0.000,C 90.000,E1 324.116} C_DIS
LIN {X 0.068,Y -522.913,Z 1188.595,A 0.000,B 0.000,C 90.000,E1 323.130} C_DIS
LIN {X 0.108,Y -520.700,Z 1188.594,A 0.000,B 0.000,C 90.000,E1 322.844} C_DIS
LIN {X 0.195,Y -517.784,Z 1188.591,A 0.000,B 0.000,C 90.000,E1 322.396} C_DIS
LIN {X 0.309,Y -515.336,Z 1188.589,A 0.000,B 0.000,C 90.000,E1 321.904} C_DIS
LIN {X 0.134,Y -513.696,Z 1188.585,A 0.000,B 0.000,C 90.000,E1 321.331} C_DIS
LIN {X 0.024,Y -512.908,Z 1188.580,A 0.000,B 0.000,C 90.000,E1 320.312} C_DIS
LIN {X -0.033,Y -513.418,Z 1188.573,A 0.000,B 0.000,C 90.000,E1 319.138} C_DIS
LIN {X 0.056,Y -514.003,Z 1188.568,A 0.000,B 0.000,C 90.000,E1 318.243} C_DIS
LIN {X 0.029,Y -514.683,Z 1188.562,A 0.000,B 0.000,C 90.000,E1 317.067} C_DIS
LIN {X 0.092,Y -515.843,Z 1188.550,A 0.000,B 0.000,C 90.000,E1 315.000} C_DIS
LIN {X -0.008,Y -516.713,Z 1188.542,A 0.000,B 0.000,C 90.000,E1 313.542} C_DIS
LIN {X -0.325,Y -518.127,Z 1188.529,A 0.000,B 0.000,C 90.000,E1 311.229} C_DIS
LIN {X 0.093,Y -518.862,Z 1188.522,A 0.000,B 0.000,C 90.000,E1 310.011} C_DIS
LIN {X 0.131,Y -519.801,Z 1188.514,A 0.000,B 0.000,C 90.000,E1 308.543} C_DIS
LIN {X 0.185,Y -520.643,Z 1188.506,A 0.000,B 0.000,C 90.000,E1 307.076} C_DIS
LIN {X 0.308,Y -521.576,Z 1188.496,A 0.000,B 0.000,C 90.000,E1 305.311} C_DIS
LIN {X -0.232,Y -522.310,Z 1188.488,A 0.000,B 0.000,C 90.000,E1 303.913} C_DIS
LIN {X 0.060,Y -523.166,Z 1188.479,A 0.000,B 0.000,C 90.000,E1 302.133} C_DIS
LIN {X 0.145,Y -523.812,Z 1188.471,A 0.000,B 0.000,C 90.000,E1 300.669} C_DIS
LIN {X 0.241,Y -524.214,Z 1188.462,A 0.000,B 0.000,C 90.000,E1 299.205} C_DIS
LIN {X 0.084,Y -524.536,Z 1188.454,A 0.000,B 0.000,C 90.000,E1 297.769} C_DIS
LIN {X 0.161,Y -524.755,Z 1188.446,A 0.000,B 0.000,C 90.000,E1 296.309} C_DIS
LIN {X -0.227,Y -524.836,Z 1188.438,A 0.000,B 0.000,C 90.000,E1 294.899} C_DIS
LIN {X 0.013,Y -524.737,Z 1188.429,A 0.000,B 0.000,C 90.000,E1 293.131} C_DIS
LIN {X -0.163,Y -524.617,Z 1188.419,A 0.000,B 0.000,C 90.000,E1 291.408} C_DIS
LIN {X 0.152,Y -524.427,Z 1188.409,A 0.000,B 0.000,C 90.000,E1 289.631} C_DIS
LIN {X -0.030,Y -524.294,Z 1188.404,A 0.000,B 0.000,C 90.000,E1 288.779} C_DIS
LIN {X -0.066,Y -523.821,Z 1188.396,A 0.000,B 0.000,C 90.000,E1 287.330} C_DIS
LIN {X 0.236,Y -523.071,Z 1188.388,A 0.000,B 0.000,C 90.000,E1 285.843} C_DIS
LIN {X 0.024,Y -521.778,Z 1188.377,A 0.000,B 0.000,C 90.000,E1 283.828} C_DIS
LIN {X 0.162,Y -520.338,Z 1188.366,A 0.000,B 0.000,C 90.000,E1 281.771} C_DIS
LIN {X 0.158,Y -519.423,Z 1188.357,A 0.000,B 0.000,C 90.000,E1 280.310} C_DIS
LIN {X 0.046,Y -518.689,Z 1188.349,A 0.000,B 0.000,C 90.000,E1 278.859} C_DIS
LIN {X -0.178,Y -517.627,Z 1188.338,A 0.000,B 0.000,C 90.000,E1 276.834} C_DIS
LIN {X 0.143,Y -516.855,Z 1188.331,A 0.000,B 0.000,C 90.000,E1 275.625} C_DIS
LIN {X 0.199,Y -515.485,Z 1188.318,A 0.000,B 0.000,C 90.000,E1 273.269} C_DIS
LIN {X 0.181,Y -514.285,Z 1188.305,A 0.000,B 0.000,C 90.000,E1 270.917} C_DIS
LIN {X -0.188,Y -513.611,Z 1188.297,A 0.000,B 0.000,C 90.000,E1 269.484} C_DIS
LIN {X 0.019,Y -513.040,Z 1188.291,A 0.000,B 0.000,C 90.000,E1 268.282} C_DIS
LIN {X 0.175,Y -512.087,Z 1188.282,A 0.000,B 0.000,C 90.000,E1 266.788} C_DIS
LIN {X -0.226,Y -511.043,Z 1188.274,A 0.000,B 0.000,C 90.000,E1 265.355} C_DIS
LIN {X -0.009,Y -510.036,Z 1188.268,A 0.000,B 0.000,C 90.000,E1 264.147} C_DIS
LIN {X 0.047,Y -508.112,Z 1188.256,A 0.000,B 0.000,C 90.000,E1 262.064} C_DIS
LIN {X 0.053,Y -506.306,Z 1188.244,A 0.000,B 0.000,C 90.000,E1 259.982} C_DIS
LIN {X 0.233,Y -504.892,Z 1188.234,A 0.000,B 0.000,C 90.000,E1 258.173} C_DIS
LIN {X -0.008,Y -503.366,Z 1188.224,A 0.000,B 0.000,C 90.000,E1 256.408} C_DIS
LIN {X -0.228,Y -501.612,Z 1188.213,A 0.000,B 0.000,C 90.000,E1 254.338} C_DIS
LIN {X 0.169,Y -499.752,Z 1188.200,A 0.000,B 0.000,C 90.000,E1 251.891} C_DIS
LIN {X -0.210,Y -498.772,Z 1188.193,A 0.000,B 0.000,C 90.000,E1 250.732} C_DIS
LIN {X -0.009,Y -497.195,Z 1188.183,A 0.000,B 0.000,C 90.000,E1 248.901} C_DIS
LIN {X -0.127,Y -495.450,Z 1188.173,A 0.000,B 0.000,C 90.000,E1 247.102} C_DIS
LIN {X 0.322,Y -493.942,Z 1188.164,A 0.000,B 0.000,C 90.000,E1 245.537} C_DIS
LIN {X 0.038,Y -492.627,Z 1188.158,A 0.000,B 0.000,C 90.000,E1 244.357} C_DIS
LIN {X 0.159,Y -491.257,Z 1188.151,A 0.000,B 0.000,C 90.000,E1 243.127} C_DIS
LIN {X 0.264,Y -489.724,Z 1188.144,A 0.000,B 0.000,C 90.000,E1 241.897} C_DIS
LIN {X 0.159,Y -487.365,Z 1188.134,A 0.000,B 0.000,C 90.000,E1 240.078} C_DIS
LIN {X 0.253,Y -485.388,Z 1188.125,A 0.000,B 0.000,C 90.000,E1 238.535} C_DIS
LIN {X 0.121,Y -482.908,Z 1188.115,A 0.000,B 0.000,C 90.000,E1 236.707} C_DIS
LIN {X -0.201,Y -480.417,Z 1188.105,A 0.000,B 0.000,C 90.000,E1 234.895} C_DIS
LIN {X -0.100,Y -478.453,Z 1188.096,A 0.000,B 0.000,C 90.000,E1 233.336} C_DIS
LIN {X -0.158,Y -475.655,Z 1188.084,A 0.000,B 0.000,C 90.000,E1 231.170} C_DIS
LIN {X -0.148,Y -473.340,Z 1188.074,A 0.000,B 0.000,C 90.000,E1 229.299} C_DIS
LIN {X 0.029,Y -471.331,Z 1188.065,A 0.000,B 0.000,C 90.000,E1 227.715} C_DIS
LIN {X -0.140,Y -467.342,Z 1188.048,A 0.000,B 0.000,C 90.000,E1 224.595} C_DIS
LIN {X 0.081,Y -464.847,Z 1188.034,A 0.000,B 0.000,C 90.000,E1 222.043} C_DIS
LIN {X 0.203,Y -463.383,Z 1188.014,A 0.000,B 0.000,C 90.000,E1 218.543} C_DIS
LIN {X -0.104,Y -463.308,Z 1188.005,A 0.000,B 0.000,C 90.000,E1 216.996} C_DIS
LIN {X -0.198,Y -463.226,Z 1187.995,A 0.000,B 0.000,C 90.000,E1 215.105} C_DIS
LIN {X 0.118,Y -464.137,Z 1187.979,A 0.000,B 0.000,C 90.000,E1 212.212} C_DIS
LIN {X -0.063,Y -465.545,Z 1187.969,A 0.000,B 0.000,C 90.000,E1 210.335} C_DIS
LIN {X -0.073,Y -468.549,Z 1187.951,A 0.000,B 0.000,C 90.000,E1 207.180} C_DIS
LIN {X 0.142,Y -473.254,Z 1187.930,A 0.000,B 0.000,C 90.000,E1 203.387} C_DIS
LIN {X -0.146,Y -479.936,Z 1187.909,A 0.000,B 0.000,C 90.000,E1 199.685} C_DIS
LIN {X 0.021,Y -489.025,Z 1187.889,A 0.000,B 0.000,C 90.000,E1 195.969} C_DIS
LIN {X -0.087,Y -497.093,Z 1187.874,A 0.000,B 0.000,C 90.000,E1 193.244} C_DIS
LIN {X 0.037,Y -502.800,Z 1187.864,A 0.000,B 0.000,C 90.000,E1 191.422} C_DIS
LIN {X 0.136,Y -509.658,Z 1187.852,A 0.000,B 0.000,C 90.000,E1 189.321} C_DIS
LIN {X -0.101,Y -513.708,Z 1187.845,A 0.000,B 0.000,C 90.000,E1 188.163} C_DIS
LIN {X 0.146,Y -518.683,Z 1187.837,A 0.000,B 0.000,C 90.000,E1 186.663} C_DIS
LIN {X -0.031,Y -523.547,Z 1187.829,A 0.000,B 0.000,C 90.000,E1 185.220} C_DIS
LIN {X -0.205,Y -529.486,Z 1187.819,A 0.000,B 0.000,C 90.000,E1 183.498} C_DIS
LIN {X -0.263,Y -536.288,Z 1187.808,A 0.000,B 0.000,C 90.000,E1 181.489} C_DIS
LIN {X -0.153,Y -543.993,Z 1187.796,A 0.000,B 0.000,C 90.000,E1 179.198} C_DIS
LIN {X 0.093,Y -549.769,Z 1187.786,A 0.000,B 0.000,C 90.000,E1 177.478} C_DIS
LIN {X -0.157,Y -554.442,Z 1187.778,A 0.000,B 0.000,C 90.000,E1 176.102} C_DIS
LIN {X 0.193,Y -558.225,Z 1187.772,A 0.000,B 0.000,C 90.000,E1 174.951} C_DIS
LIN {X 0.274,Y -563.678,Z 1187.763,A 0.000,B 0.000,C 90.000,E1 173.280} C_DIS
LIN {X -0.020,Y -569.094,Z 1187.754,A 0.000,B 0.000,C 90.000,E1 171.659} C_DIS
LIN {X 0.064,Y -572.672,Z 1187.748,A 0.000,B 0.000,C 90.000,E1 170.557} C_DIS
LIN {X -0.162,Y -577.085,Z 1187.740,A 0.000,B 0.000,C 90.000,E1 169.218} C_DIS
LIN {X 0.132,Y -583.165,Z 1187.729,A 0.000,B 0.000,C 90.000,E1 167.297} C_DIS
LIN {X -0.244,Y -587.536,Z 1187.722,A 0.000,B 0.000,C 90.000,E1 165.992} C_DIS
LIN {X 0.035,Y -591.826,Z 1187.715,A 0.000,B 0.000,C 90.000,E1 164.629} C_DIS
LIN {X -0.039,Y -597.776,Z 1187.704,A 0.000,B 0.000,C 90.000,E1 162.779} C_DIS
LIN {X -0.168,Y -600.340,Z 1187.700,A 0.000,B 0.000,C 90.000,E1 162.000} C_DIS
LIN {X -0.080,Y -604.519,Z 1187.693,A 0.000,B 0.000,C 90.000,E1 160.678} C_DIS
LIN {X 0.217,Y -609.376,Z 1187.684,A 0.000,B 0.000,C 90.000,E1 159.082} C_DIS
LIN {X 0.051,Y -614.121,Z 1187.675,A 0.000,B 0.000,C 90.000,E1 157.539} C_DIS
LIN {X 0.240,Y -618.033,Z 1187.668,A 0.000,B 0.000,C 90.000,E1 156.230} C_DIS
LIN {X -0.066,Y -621.133,Z 1187.662,A 0.000,B 0.000,C 90.000,E1 155.229} C_DIS
LIN {X -0.063,Y -624.823,Z 1187.655,A 0.000,B 0.000,C 90.000,E1 153.948} C_DIS
LIN {X 0.028,Y -629.069,Z 1187.647,A 0.000,B 0.000,C 90.000,E1 152.410} C_DIS
LIN {X 0.159,Y -632.504,Z 1187.640,A 0.000,B 0.000,C 90.000,E1 151.129} C_DIS
LIN {X 0.131,Y -636.432,Z 1187.631,A 0.000,B 0.000,C 90.000,E1 149.616} C_DIS
LIN {X -0.086,Y -639.474,Z 1187.624,A 0.000,B 0.000,C 90.000,E1 148.377} C_DIS
LIN {X -0.042,Y -642.348,Z 1187.617,A 0.000,B 0.000,C 90.000,E1 147.120} C_DIS
LIN {X 0.330,Y -644.529,Z 1187.612,A 0.000,B 0.000,C 90.000,E1 146.087} C_DIS
LIN {X 0.149,Y -647.530,Z 1187.604,A 0.000,B 0.000,C 90.000,E1 144.609} C_DIS
LIN {X -0.410,Y -649.840,Z 1187.597,A 0.000,B 0.000,C 90.000,E1 143.417} C_DIS
LIN {X -0.033,Y -652.089,Z 1187.590,A 0.000,B 0.000,C 90.000,E1 142.145} C_DIS
LIN {X 0.197,Y -655.789,Z 1187.579,A 0.000,B 0.000,C 90.000,E1 140.150} C_DIS
LIN {X 0.062,Y -658.272,Z 1187.572,A 0.000,B 0.000,C 90.000,E1 138.933} C_DIS
LIN {X -0.055,Y -661.463,Z 1187.564,A 0.000,B 0.000,C 90.000,E1 137.472} C_DIS
LIN {X 0.341,Y -664.549,Z 1187.556,A 0.000,B 0.000,C 90.000,E1 135.972} C_DIS
LIN {X 0.331,Y -668.801,Z 1187.545,A 0.000,B 0.000,C 90.000,E1 134.028} C_DIS
LIN {X -0.027,Y -673.973,Z 1187.533,A 0.000,B 0.000,C 90.000,E1 131.881} C_DIS
LIN {X 0.255,Y -677.992,Z 1187.523,A 0.000,B 0.000,C 90.000,E1 130.172} C_DIS
LIN {X 0.053,Y -680.988,Z 1187.517,A 0.000,B 0.000,C 90.000,E1 128.991} C_DIS
LIN {X 0.087,Y -685.139,Z 1187.507,A 0.000,B 0.000,C 90.000,E1 127.317} C_DIS
LIN {X 0.167,Y -688.731,Z 1187.500,A 0.000,B 0.000,C 90.000,E1 125.884} C_DIS
LIN {X 0.031,Y -690.473,Z 1187.495,A 0.000,B 0.000,C 90.000,E1 125.185} C_DIS
LIN {X -0.195,Y -693.771,Z 1187.488,A 0.000,B 0.000,C 90.000,E1 123.785} C_DIS
LIN {X -0.291,Y -695.366,Z 1187.484,A 0.000,B 0.000,C 90.000,E1 123.086} C_DIS
LIN {X 0.109,Y -697.895,Z 1187.477,A 0.000,B 0.000,C 90.000,E1 121.878} C_DIS
LIN {X 0.218,Y -700.677,Z 1187.469,A 0.000,B 0.000,C 90.000,E1 120.463} C_DIS
LIN {X -0.258,Y -702.727,Z 1187.463,A 0.000,B 0.000,C 90.000,E1 119.333} C_DIS
LIN {X -0.095,Y -704.550,Z 1187.456,A 0.000,B 0.000,C 90.000,E1 118.153} C_DIS
LIN {X -0.187,Y -705.525,Z 1187.453,A 0.000,B 0.000,C 90.000,E1 117.462} C_DIS
LIN {X 0.058,Y -706.162,Z 1187.449,A 0.000,B 0.000,C 90.000,E1 116.744} C_DIS
LIN {X -0.347,Y -706.645,Z 1187.443,A 0.000,B 0.000,C 90.000,E1 115.848} C_DIS
LIN {X -0.405,Y -706.701,Z 1187.440,A 0.000,B 0.000,C 90.000,E1 115.155} C_DIS
LIN {X 0.183,Y -706.470,Z 1187.437,A 0.000,B 0.000,C 90.000,E1 114.643} C_DIS
LIN {X -0.460,Y -706.196,Z 1187.436,A 0.000,B 0.000,C 90.000,E1 114.463} C_DIS
LIN {X 0.123,Y -705.326,Z 1187.433,A 0.000,B 0.000,C 90.000,E1 113.951} C_DIS
LIN {X 0.126,Y -704.415,Z 1187.432,A 0.000,B 0.000,C 90.000,E1 113.718} C_DIS
LIN {X 0.049,Y -702.153,Z 1187.429,A 0.000,B 0.000,C 90.000,E1 113.259} C_DIS
LIN {X 0.186,Y -701.192,Z 1187.429,A 0.000,B 0.000,C 90.000,E1 113.131} C_DIS
LIN {X 0.004,Y -696.087,Z 1187.426,A 0.000,B 0.000,C 90.000,E1 112.695} C_DIS
LIN {X -0.057,Y -694.389,Z 1187.426,A 0.000,B 0.000,C 90.000,E1 112.589} C_DIS
LIN {X -0.292,Y -691.872,Z 1187.425,A 0.000,B 0.000,C 90.000,E1 112.514} C_DIS
LIN {X 0.112,Y -687.047,Z 1187.424,A 0.000,B 0.000,C 90.000,E1 112.333} C_DIS
LIN {X 0.112,Y -684.813,Z 1187.424,A 0.000,B 0.000,C 90.000,E1 112.280} C_DIS
LIN {X -0.255,Y -677.801,Z 1187.424,A 0.000,B 0.000,C 90.000,E1 112.280} C_DIS
LIN {X -0.059,Y -606.586,Z 1187.424,A 0.000,B 0.000,C 90.000,E1 112.259} C_DIS
LIN {X 0.087,Y -601.433,Z 1187.422,A 0.000,B 0.000,C 90.000,E1 111.897} C_DIS
LIN {X 0.356,Y -590.386,Z 1187.417,A 0.000,B 0.000,C 90.000,E1 110.972} C_DIS
LIN {X -0.033,Y -580.673,Z 1187.412,A 0.000,B 0.000,C 90.000,E1 110.248} C_DIS
LIN {X -0.015,Y -571.732,Z 1187.409,A 0.000,B 0.000,C 90.000,E1 109.577} C_DIS
LIN {X 0.144,Y -562.782,Z 1187.405,A 0.000,B 0.000,C 90.000,E1 108.906} C_DIS
LIN {X 0.268,Y -558.973,Z 1187.404,A 0.000,B 0.000,C 90.000,E1 108.598} C_DIS
LIN {X -0.004,Y -558.158,Z 1187.403,A 0.000,B 0.000,C 90.000,E1 108.544} C_DIS
LIN {X -0.123,Y -555.734,Z 1187.401,A 0.000,B 0.000,C 90.000,E1 108.236} C_DIS
LIN {X 0.284,Y -555.064,Z 1187.401,A 0.000,B 0.000,C 90.000,E1 108.055} C_DIS
LIN {X -0.007,Y -554.380,Z 1187.399,A 0.000,B 0.000,C 90.000,E1 107.764} C_DIS
LIN {X 0.129,Y -552.950,Z 1187.394,A 0.000,B 0.000,C 90.000,E1 106.913} C_DIS
LIN {X -0.206,Y -552.781,Z 1187.393,A 0.000,B 0.000,C 90.000,E1 106.677} C_DIS
LIN {X -0.249,Y -552.797,Z 1187.393,A 0.000,B 0.000,C 90.000,E1 106.677} C_DIS
LIN {X -0.159,Y -553.401,Z 1187.392,A 0.000,B 0.000,C 90.000,E1 106.496} C_DIS
LIN {X 0.086,Y -553.824,Z 1187.389,A 0.000,B 0.000,C 90.000,E1 106.024} C_DIS
LIN {X -0.332,Y -553.780,Z 1187.388,A 0.000,B 0.000,C 90.000,E1 105.788} C_DIS
LIN {X 0.069,Y -553.902,Z 1187.387,A 0.000,B 0.000,C 90.000,E1 105.607} C_DIS
LIN {X -0.066,Y -554.174,Z 1187.386,A 0.000,B 0.000,C 90.000,E1 105.481} C_DIS
LIN {X 0.174,Y -554.269,Z 1187.383,A 0.000,B 0.000,C 90.000,E1 104.898} C_DIS
LIN {X -0.269,Y -554.367,Z 1187.382,A 0.000,B 0.000,C 90.000,E1 104.773} C_DIS
LIN {X -0.147,Y -555.226,Z 1187.380,A 0.000,B 0.000,C 90.000,E1 104.481} C_DIS
LIN {X -0.161,Y -555.113,Z 1187.378,A 0.000,B 0.000,C 90.000,E1 104.064} C_DIS
LIN {X 0.239,Y -555.404,Z 1187.377,A 0.000,B 0.000,C 90.000,E1 103.883} C_DIS
LIN {X -0.174,Y -555.513,Z 1187.376,A 0.000,B 0.000,C 90.000,E1 103.647} C_DIS
LIN {X -0.044,Y -555.085,Z 1187.374,A 0.000,B 0.000,C 90.000,E1 103.355} C_DIS
LIN {X 0.220,Y -555.234,Z 1187.372,A 0.000,B 0.000,C 90.000,E1 102.883} C_DIS
LIN {X -0.047,Y -555.041,Z 1187.371,A 0.000,B 0.000,C 90.000,E1 102.771} C_DIS
LIN {X -0.084,Y -555.297,Z 1187.368,A 0.000,B 0.000,C 90.000,E1 102.187} C_DIS
LIN {X -0.107,Y -557.285,Z 1187.355,A 0.000,B 0.000,C 90.000,E1 99.962} C_DIS
LIN {X -0.200,Y -558.355,Z 1187.349,A 0.000,B 0.000,C 90.000,E1 98.859} C_DIS
LIN {X -0.140,Y -559.654,Z 1187.341,A 0.000,B 0.000,C 90.000,E1 97.466} C_DIS
LIN {X 0.280,Y -560.622,Z 1187.335,A 0.000,B 0.000,C 90.000,E1 96.315} C_DIS
LIN {X 0.248,Y -561.629,Z 1187.328,A 0.000,B 0.000,C 90.000,E1 94.935} C_DIS
LIN {X -0.102,Y -562.920,Z 1187.317,A 0.000,B 0.000,C 90.000,E1 93.037} C_DIS
LIN {X -0.030,Y -564.098,Z 1187.308,A 0.000,B 0.000,C 90.000,E1 91.375} C_DIS
LIN {X 0.060,Y -565.356,Z 1187.298,A 0.000,B 0.000,C 90.000,E1 89.714} C_DIS
LIN {X -0.261,Y -566.688,Z 1187.288,A 0.000,B 0.000,C 90.000,E1 87.822} C_DIS
LIN {X 0.231,Y -567.470,Z 1187.282,A 0.000,B 0.000,C 90.000,E1 86.674} C_DIS
LIN {X -0.288,Y -568.458,Z 1187.274,A 0.000,B 0.000,C 90.000,E1 85.355} C_DIS
LIN {X 0.157,Y -569.815,Z 1187.263,A 0.000,B 0.000,C 90.000,E1 83.394} C_DIS
LIN {X -0.110,Y -570.932,Z 1187.254,A 0.000,B 0.000,C 90.000,E1 81.781} C_DIS
LIN {X -0.013,Y -571.619,Z 1187.248,A 0.000,B 0.000,C 90.000,E1 80.679} C_DIS
LIN {X -0.277,Y -572.409,Z 1187.241,A 0.000,B 0.000,C 90.000,E1 79.342} C_DIS
LIN {X 0.143,Y -573.178,Z 1187.233,A 0.000,B 0.000,C 90.000,E1 77.937} C_DIS
LIN {X 0.016,Y -573.881,Z 1187.226,A 0.000,B 0.000,C 90.000,E1 76.589} C_DIS
LIN {X 0.027,Y -574.891,Z 1187.215,A 0.000,B 0.000,C 90.000,E1 74.685} C_DIS
LIN {X 0.079,Y -576.151,Z 1187.201,A 0.000,B 0.000,C 90.000,E1 72.236} C_DIS
LIN {X -0.237,Y -577.298,Z 1187.191,A 0.000,B 0.000,C 90.000,E1 70.369} C_DIS
LIN {X 0.118,Y -579.693,Z 1187.174,A 0.000,B 0.000,C 90.000,E1 67.358} C_DIS
LIN {X -0.293,Y -581.049,Z 1187.167,A 0.000,B 0.000,C 90.000,E1 66.049} C_DIS
LIN {X -0.180,Y -582.795,Z 1187.156,A 0.000,B 0.000,C 90.000,E1 64.152} C_DIS
LIN {X 0.106,Y -584.946,Z 1187.144,A 0.000,B 0.000,C 90.000,E1 61.975} C_DIS
LIN {X -0.231,Y -586.202,Z 1187.137,A 0.000,B 0.000,C 90.000,E1 60.667} C_DIS
LIN {X -0.255,Y -587.377,Z 1187.130,A 0.000,B 0.000,C 90.000,E1 59.331} C_DIS
LIN {X -0.257,Y -588.487,Z 1187.122,A 0.000,B 0.000,C 90.000,E1 57.995} C_DIS
LIN {X 0.075,Y -589.487,Z 1187.115,A 0.000,B 0.000,C 90.000,E1 56.628} C_DIS
LIN {X 0.007,Y -590.870,Z 1187.104,A 0.000,B 0.000,C 90.000,E1 54.769} C_DIS
LIN {X -0.033,Y -591.976,Z 1187.095,A 0.000,B 0.000,C 90.000,E1 53.176} C_DIS
LIN {X 0.023,Y -593.343,Z 1187.084,A 0.000,B 0.000,C 90.000,E1 51.045} C_DIS
LIN {X 0.157,Y -594.276,Z 1187.073,A 0.000,B 0.000,C 90.000,E1 49.175} C_DIS
LIN {X -0.118,Y -594.715,Z 1187.066,A 0.000,B 0.000,C 90.000,E1 47.877} C_DIS
LIN {X 0.035,Y -594.923,Z 1187.062,A 0.000,B 0.000,C 90.000,E1 47.067} C_DIS
LIN {X 0.176,Y -594.950,Z 1187.054,A 0.000,B 0.000,C 90.000,E1 45.729} C_DIS
LIN {X -0.110,Y -594.849,Z 1187.047,A 0.000,B 0.000,C 90.000,E1 44.433} C_DIS
LIN {X -0.176,Y -594.478,Z 1187.041,A 0.000,B 0.000,C 90.000,E1 43.380} C_DIS
LIN {X 0.009,Y -594.020,Z 1187.036,A 0.000,B 0.000,C 90.000,E1 42.567} C_DIS
LIN {X 0.131,Y -593.160,Z 1187.029,A 0.000,B 0.000,C 90.000,E1 41.229} C_DIS
LIN {X -0.134,Y -592.527,Z 1187.025,A 0.000,B 0.000,C 90.000,E1 40.458} C_DIS
LIN {X 0.045,Y -591.857,Z 1187.020,A 0.000,B 0.000,C 90.000,E1 39.644} C_DIS
LIN {X -0.034,Y -590.809,Z 1187.014,A 0.000,B 0.000,C 90.000,E1 38.588} C_DIS
LIN {X -0.240,Y -589.866,Z 1187.010,A 0.000,B 0.000,C 90.000,E1 37.810} C_DIS
LIN {X -0.044,Y -587.895,Z 1187.003,A 0.000,B 0.000,C 90.000,E1 36.457} C_DIS
LIN {X 0.074,Y -586.590,Z 1186.998,A 0.000,B 0.000,C 90.000,E1 35.644} C_DIS
LIN {X 0.308,Y -584.925,Z 1186.994,A 0.000,B 0.000,C 90.000,E1 34.818} C_DIS
LIN {X 0.045,Y -583.111,Z 1186.989,A 0.000,B 0.000,C 90.000,E1 34.040} C_DIS
LIN {X -0.103,Y -582.494,Z 1186.988,A 0.000,B 0.000,C 90.000,E1 33.785} C_DIS
LIN {X 0.256,Y -579.300,Z 1186.982,A 0.000,B 0.000,C 90.000,E1 32.673} C_DIS
LIN {X 0.105,Y -576.624,Z 1186.977,A 0.000,B 0.000,C 90.000,E1 31.878} C_DIS
LIN {X -0.067,Y -573.434,Z 1186.973,A 0.000,B 0.000,C 90.000,E1 31.082} C_DIS
LIN {X 0.105,Y -570.510,Z 1186.969,A 0.000,B 0.000,C 90.000,E1 30.384} C_DIS
LIN {X -0.048,Y -567.288,Z 1186.965,A 0.000,B 0.000,C 90.000,E1 29.716} C_DIS
LIN {X -0.012,Y -563.748,Z 1186.961,A 0.000,B 0.000,C 90.000,E1 29.027} C_DIS
LIN {X 0.070,Y -558.271,Z 1186.956,A 0.000,B 0.000,C 90.000,E1 28.052} C_DIS
LIN {X -0.085,Y -554.932,Z 1186.953,A 0.000,B 0.000,C 90.000,E1 27.513} C_DIS
LIN {X -0.006,Y -549.567,Z 1186.948,A 0.000,B 0.000,C 90.000,E1 26.668} C_DIS
LIN {X 0.014,Y -545.641,Z 1186.945,A 0.000,B 0.000,C 90.000,E1 26.104} C_DIS
LIN {X -0.247,Y -539.075,Z 1186.940,A 0.000,B 0.000,C 90.000,E1 25.283} C_DIS
LIN {X 0.135,Y -532.098,Z 1186.936,A 0.000,B 0.000,C 90.000,E1 24.387} C_DIS
LIN {X -0.088,Y -525.825,Z 1186.932,A 0.000,B 0.000,C 90.000,E1 23.695} C_DIS
LIN {X 0.237,Y -519.435,Z 1186.928,A 0.000,B 0.000,C 90.000,E1 22.950} C_DIS
LIN {X -0.060,Y -512.663,Z 1186.924,A 0.000,B 0.000,C 90.000,E1 22.280} C_DIS
LIN {X -0.165,Y -504.431,Z 1186.919,A 0.000,B 0.000,C 90.000,E1 21.461} C_DIS
LIN {X 0.102,Y -494.515,Z 1186.914,A 0.000,B 0.000,C 90.000,E1 20.482} C_DIS
LIN {X 0.051,Y -485.767,Z 1186.909,A 0.000,B 0.000,C 90.000,E1 19.685} C_DIS
LIN {X -0.072,Y -476.979,Z 1186.905,A 0.000,B 0.000,C 90.000,E1 18.906} C_DIS
LIN {X -0.180,Y -468.098,Z 1186.901,A 0.000,B 0.000,C 90.000,E1 18.127} C_DIS
LIN {X -0.077,Y -450.768,Z 1186.892,A 0.000,B 0.000,C 90.000,E1 16.551} C_DIS
LIN {X 0.083,Y -429.268,Z 1186.880,A 0.000,B 0.000,C 90.000,E1 14.426} C_DIS
LIN {X 0.081,Y -415.186,Z 1186.872,A 0.000,B 0.000,C 90.000,E1 12.883} C_DIS
LIN {X 0.074,Y -403.249,Z 1186.864,A 0.000,B 0.000,C 90.000,E1 11.422} C_DIS
LIN {X -0.216,Y -398.271,Z 1186.860,A 0.000,B 0.000,C 90.000,E1 10.782} C_DIS
LIN {X -0.060,Y -396.589,Z 1186.858,A 0.000,B 0.000,C 90.000,E1 10.489} C_DIS
LIN {X 0.141,Y -394.845,Z 1186.856,A 0.000,B 0.000,C 90.000,E1 10.141} C_DIS
LIN {X -0.161,Y -393.326,Z 1186.854,A 0.000,B 0.000,C 90.000,E1 9.782} C_DIS
LIN {X 0.189,Y -393.306,Z 1186.854,A 0.000,B 0.000,C 90.000,E1 9.726} C_DIS
LIN {X -0.078,Y -393.295,Z 1186.852,A 0.000,B 0.000,C 90.000,E1 9.378} C_DIS
LIN {X 0.001,Y -394.727,Z 1186.849,A 0.000,B 0.000,C 90.000,E1 8.746} C_DIS
LIN {X 0.123,Y -397.568,Z 1186.845,A 0.000,B 0.000,C 90.000,E1 7.992} C_DIS
LIN {X 0.060,Y -400.639,Z 1186.842,A 0.000,B 0.000,C 90.000,E1 7.473} C_DIS
LIN {X 0.045,Y -402.697,Z 1186.840,A 0.000,B 0.000,C 90.000,E1 7.125} C_DIS
LIN {X -0.036,Y -405.750,Z 1186.838,A 0.000,B 0.000,C 90.000,E1 6.777} C_DIS
LIN {X 0.143,Y -409.781,Z 1186.836,A 0.000,B 0.000,C 90.000,E1 6.372} C_DIS
LIN {X -0.201,Y -413.059,Z 1186.834,A 0.000,B 0.000,C 90.000,E1 6.144} C_DIS
LIN {X 0.015,Y -425.365,Z 1186.829,A 0.000,B 0.000,C 90.000,E1 5.163} C_DIS
LIN {X 0.065,Y -439.807,Z 1186.823,A 0.000,B 0.000,C 90.000,E1 4.073} C_DIS
LIN {X -0.097,Y -459.103,Z 1186.815,A 0.000,B 0.000,C 90.000,E1 2.694} C_DIS
LIN {X -0.081,Y -466.986,Z 1186.812,A 0.000,B 0.000,C 90.000,E1 2.121} C_DIS
LIN {X -0.174,Y -474.791,Z 1186.808,A 0.000,B 0.000,C 90.000,E1 1.547} C_DIS
LIN {X 0.141,Y -483.864,Z 1186.805,A 0.000,B 0.000,C 90.000,E1 0.802} C_DIS
LIN {X 0.216,Y -491.251,Z 1186.801,A 0.000,B 0.000,C 90.000,E1 0.172} C_DIS
LIN {X 0.037,Y -497.172,Z 1186.798,A 0.000,B 0.000,C 90.000,E1 359.656} C_DIS
LIN {X 0.064,Y -504.042,Z 1186.794,A 0.000,B 0.000,C 90.000,E1 358.969} C_DIS
LIN {X 0.073,Y -511.806,Z 1186.790,A 0.000,B 0.000,C 90.000,E1 358.108} C_DIS
LIN {X -0.094,Y -516.784,Z 1186.786,A 0.000,B 0.000,C 90.000,E1 357.535} C_DIS
LIN {X 0.173,Y -522.415,Z 1186.782,A 0.000,B 0.000,C 90.000,E1 356.788} C_DIS
LIN {X -0.208,Y -527.550,Z 1186.778,A 0.000,B 0.000,C 90.000,E1 356.102} C_DIS
LIN {X -0.237,Y -531.418,Z 1186.775,A 0.000,B 0.000,C 90.000,E1 355.527} C_DIS
LIN {X 0.024,Y -535.745,Z 1186.771,A 0.000,B 0.000,C 90.000,E1 354.780} C_DIS
LIN {X 0.111,Y -540.234,Z 1186.766,A 0.000,B 0.000,C 90.000,E1 353.913} C_DIS
LIN {X 0.181,Y -543.080,Z 1186.763,A 0.000,B 0.000,C 90.000,E1 353.337} C_DIS
LIN {X 0.271,Y -545.658,Z 1186.760,A 0.000,B 0.000,C 90.000,E1 352.761} C_DIS
LIN {X 0.190,Y -548.623,Z 1186.756,A 0.000,B 0.000,C 90.000,E1 352.064} C_DIS
LIN {X -0.233,Y -550.824,Z 1186.753,A 0.000,B 0.000,C 90.000,E1 351.546} C_DIS
LIN {X 0.015,Y -553.788,Z 1186.748,A 0.000,B 0.000,C 90.000,E1 350.679} C_DIS
LIN {X 0.260,Y -555.596,Z 1186.745,A 0.000,B 0.000,C 90.000,E1 350.095} C_DIS
LIN {X 0.144,Y -558.929,Z 1186.739,A 0.000,B 0.000,C 90.000,E1 348.993} C_DIS
LIN {X 0.028,Y -561.179,Z 1186.734,A 0.000,B 0.000,C 90.000,E1 348.173} C_DIS
LIN {X 0.092,Y -563.955,Z 1186.728,A 0.000,B 0.000,C 90.000,E1 347.061} C_DIS
LIN {X -0.225,Y -566.574,Z 1186.722,A 0.000,B 0.000,C 90.000,E1 345.992} C_DIS
LIN {X 0.228,Y -569.576,Z 1186.714,A 0.000,B 0.000,C 90.000,E1 344.574} C_DIS
LIN {X -0.005,Y -571.854,Z 1186.708,A 0.000,B 0.000,C 90.000,E1 343.504} C_DIS
LIN {X -0.047,Y -575.026,Z 1186.699,A 0.000,B 0.000,C 90.000,E1 341.873} C_DIS
LIN {X 0.151,Y -577.385,Z 1186.692,A 0.000,B 0.000,C 90.000,E1 340.496} C_DIS
LIN {X -0.157,Y -578.902,Z 1186.686,A 0.000,B 0.000,C 90.000,E1 339.444} C_DIS
LIN {X 0.108,Y -580.206,Z 1186.680,A 0.000,B 0.000,C 90.000,E1 338.337} C_DIS
LIN {X 0.137,Y -580.747,Z 1186.677,A 0.000,B 0.000,C 90.000,E1 337.794} C_DIS
LIN {X -0.119,Y -581.551,Z 1186.671,A 0.000,B 0.000,C 90.000,E1 336.741} C_DIS
LIN {X 0.003,Y -581.732,Z 1186.666,A 0.000,B 0.000,C 90.000,E1 335.921} C_DIS
LIN {X 0.130,Y -581.552,Z 1186.662,A 0.000,B 0.000,C 90.000,E1 335.101} C_DIS
LIN {X -0.137,Y -581.325,Z 1186.659,A 0.000,B 0.000,C 90.000,E1 334.588} C_DIS
LIN {X -0.015,Y -580.581,Z 1186.654,A 0.000,B 0.000,C 90.000,E1 333.768} C_DIS
LIN {X -0.287,Y -579.932,Z 1186.651,A 0.000,B 0.000,C 90.000,E1 333.256} C_DIS
LIN {X -0.062,Y -577.934,Z 1186.645,A 0.000,B 0.000,C 90.000,E1 332.153} C_DIS
LIN {X 0.284,Y -576.102,Z 1186.641,A 0.000,B 0.000,C 90.000,E1 331.307} C_DIS
LIN {X -0.176,Y -573.989,Z 1186.636,A 0.000,B 0.000,C 90.000,E1 330.539} C_DIS
LIN {X -0.211,Y -572.293,Z 1186.633,A 0.000,B 0.000,C 90.000,E1 329.999} C_DIS
LIN {X 0.235,Y -570.255,Z 1186.630,A 0.000,B 0.000,C 90.000,E1 329.410} C_DIS
LIN {X 0.086,Y -567.181,Z 1186.626,A 0.000,B 0.000,C 90.000,E1 328.742} C_DIS
LIN {X -0.093,Y -563.338,Z 1186.623,A 0.000,B 0.000,C 90.000,E1 328.074} C_DIS
LIN {X -0.114,Y -557.871,Z 1186.618,A 0.000,B 0.000,C 90.000,E1 327.248} C_DIS
LIN {X -0.145,Y -554.927,Z 1186.616,A 0.000,B 0.000,C 90.000,E1 326.834} C_DIS
LIN {X -0.206,Y -548.508,Z 1186.611,A 0.000,B 0.000,C 90.000,E1 326.008} C_DIS
LIN {X 0.205,Y -542.766,Z 1186.607,A 0.000,B 0.000,C 90.000,E1 325.261} C_DIS
LIN {X 0.122,Y -534.117,Z 1186.602,A 0.000,B 0.000,C 90.000,E1 324.276} C_DIS
LIN {X 0.198,Y -524.092,Z 1186.595,A 0.000,B 0.000,C 90.000,E1 323.130} C_DIS
LIN {X 0.225,Y -521.744,Z 1186.594,A 0.000,B 0.000,C 90.000,E1 322.844} C_DIS
LIN {X -0.164,Y -518.357,Z 1186.591,A 0.000,B 0.000,C 90.000,E1 322.396} C_DIS
LIN {X -0.072,Y -515.816,Z 1186.588,A 0.000,B 0.000,C 90.000,E1 321.904} C_DIS
LIN {X -0.053,Y -514.054,Z 1186.585,A 0.000,B 0.000,C 90.000,E1 321.295} C_DIS
LIN {X -0.278,Y -513.317,Z 1186.580,A 0.000,B 0.000,C 90.000,E1 320.436} C_DIS
LIN {X -0.028,Y -513.250,Z 1186.578,A 0.000,B 0.000,C 90.000,E1 320.114} C_DIS
LIN {X 0.066,Y -513.646,Z 1186.573,A 0.000,B 0.000,C 90.000,E1 319.218} C_DIS
LIN {X 0.158,Y -514.302,Z 1186.569,A 0.000,B 0.000,C 90.000,E1 318.324} C_DIS
LIN {X 0.048,Y -515.118,Z 1186.560,A 0.000,B 0.000,C 90.000,E1 316.863} C_DIS
LIN {X -0.255,Y -516.295,Z 1186.549,A 0.000,B 0.000,C 90.000,E1 314.838} C_DIS
LIN {X 0.029,Y -517.180,Z 1186.541,A 0.000,B 0.000,C 90.000,E1 313.338} C_DIS
LIN {X -0.197,Y -518.383,Z 1186.529,A 0.000,B 0.000,C 90.000,E1 311.310} C_DIS
LIN {X 0.166,Y -519.326,Z 1186.521,A 0.000,B 0.000,C 90.000,E1 309.806} C_DIS
LIN {X -0.190,Y -520.238,Z 1186.513,A 0.000,B 0.000,C 90.000,E1 308.382} C_DIS
LIN {X -0.082,Y -520.945,Z 1186.507,A 0.000,B 0.000,C 90.000,E1 307.202} C_DIS
LIN {X -0.008,Y -522.060,Z 1186.495,A 0.000,B 0.000,C 90.000,E1 305.152} C_DIS
LIN {X -0.111,Y -522.771,Z 1186.487,A 0.000,B 0.000,C 90.000,E1 303.706} C_DIS
LIN {X -0.137,Y -523.820,Z 1186.476,A 0.000,B 0.000,C 90.000,E1 301.671} C_DIS
LIN {X -0.115,Y -524.215,Z 1186.471,A 0.000,B 0.000,C 90.000,E1 300.797} C_DIS
LIN {X 0.129,Y -524.686,Z 1186.461,A 0.000,B 0.000,C 90.000,E1 299.027} C_DIS
LIN {X -0.012,Y -525.028,Z 1186.453,A 0.000,B 0.000,C 90.000,E1 297.590} C_DIS
LIN {X -0.159,Y -525.229,Z 1186.445,A 0.000,B 0.000,C 90.000,E1 296.155} C_DIS
LIN {X -0.074,Y -525.301,Z 1186.437,A 0.000,B 0.000,C 90.000,E1 294.695} C_DIS
LIN {X -0.040,Y -525.166,Z 1186.427,A 0.000,B 0.000,C 90.000,E1 292.950} C_DIS
LIN {X 0.118,Y -525.057,Z 1186.419,A 0.000,B 0.000,C 90.000,E1 291.482} C_DIS
LIN {X -0.208,Y -524.883,Z 1186.411,A 0.000,B 0.000,C 90.000,E1 290.066} C_DIS
LIN {X -0.216,Y -524.749,Z 1186.405,A 0.000,B 0.000,C 90.000,E1 288.906} C_DIS
LIN {X -0.240,Y -524.337,Z 1186.397,A 0.000,B 0.000,C 90.000,E1 287.457} C_DIS
LIN {X 0.076,Y -523.605,Z 1186.389,A 0.000,B 0.000,C 90.000,E1 285.969} C_DIS
LIN {X 0.014,Y -522.364,Z 1186.377,A 0.000,B 0.000,C 90.000,E1 283.939} C_DIS
LIN {X 0.157,Y -520.907,Z 1186.366,A 0.000,B 0.000,C 90.000,E1 281.883} C_DIS
LIN {X 0.063,Y -519.983,Z 1186.358,A 0.000,B 0.000,C 90.000,E1 280.433} C_DIS
LIN {X 0.052,Y -519.252,Z 1186.350,A 0.000,B 0.000,C 90.000,E1 278.973} C_DIS
LIN {X -0.163,Y -518.175,Z 1186.339,A 0.000,B 0.000,C 90.000,E1 276.947} C_DIS
LIN {X 0.090,Y -517.211,Z 1186.330,A 0.000,B 0.000,C 90.000,E1 275.454} C_DIS
LIN {X 0.191,Y -515.861,Z 1186.317,A 0.000,B 0.000,C 90.000,E1 273.094} C_DIS
LIN {X 0.086,Y -514.568,Z 1186.303,A 0.000,B 0.000,C 90.000,E1 270.458} C_DIS
LIN {X 0.236,Y -513.873,Z 1186.294,A 0.000,B 0.000,C 90.000,E1 268.969} C_DIS
LIN {X 0.026,Y -513.418,Z 1186.290,A 0.000,B 0.000,C 90.000,E1 268.108} C_DIS
LIN {X 0.170,Y -512.492,Z 1186.281,A 0.000,B 0.000,C 90.000,E1 266.617} C_DIS
LIN {X -0.185,Y -511.428,Z 1186.273,A 0.000,B 0.000,C 90.000,E1 265.179} C_DIS
LIN {X 0.046,Y -510.381,Z 1186.267,A 0.000,B 0.000,C 90.000,E1 263.970} C_DIS
LIN {X 0.099,Y -508.764,Z 1186.257,A 0.000,B 0.000,C 90.000,E1 262.186} C_DIS
LIN {X 0.197,Y -506.953,Z 1186.245,A 0.000,B 0.000,C 90.000,E1 260.095} C_DIS
LIN {X -0.100,Y -505.507,Z 1186.235,A 0.000,B 0.000,C 90.000,E1 258.342} C_DIS
LIN {X 0.115,Y -503.705,Z 1186.224,A 0.000,B 0.000,C 90.000,E1 256.228} C_DIS
LIN {X -0.093,Y -501.970,Z 1186.212,A 0.000,B 0.000,C 90.000,E1 254.157} C_DIS
LIN {X -0.070,Y -500.344,Z 1186.200,A 0.000,B 0.000,C 90.000,E1 252.054} C_DIS
LIN {X -0.059,Y -499.084,Z 1186.192,A 0.000,B 0.000,C 90.000,E1 250.550} C_DIS
LIN {X 0.146,Y -497.432,Z 1186.182,A 0.000,B 0.000,C 90.000,E1 248.720} C_DIS
LIN {X -0.023,Y -496.013,Z 1186.174,A 0.000,B 0.000,C 90.000,E1 247.230} C_DIS
LIN {X -0.220,Y -494.527,Z 1186.165,A 0.000,B 0.000,C 90.000,E1 245.741} C_DIS
LIN {X -0.035,Y -492.816,Z 1186.157,A 0.000,B 0.000,C 90.000,E1 244.204} C_DIS
LIN {X -0.125,Y -491.435,Z 1186.150,A 0.000,B 0.000,C 90.000,E1 242.999} C_DIS
LIN {X -0.015,Y -489.870,Z 1186.143,A 0.000,B 0.000,C 90.000,E1 241.769} C_DIS
LIN {X -0.116,Y -487.909,Z 1186.135,A 0.000,B 0.000,C 90.000,E1 240.255} C_DIS
LIN {X -0.255,Y -485.927,Z 1186.126,A 0.000,B 0.000,C 90.000,E1 238.742} C_DIS
LIN {X 0.295,Y -483.398,Z 1186.116,A 0.000,B 0.000,C 90.000,E1 236.834} C_DIS
LIN {X 0.173,Y -481.284,Z 1186.107,A 0.000,B 0.000,C 90.000,E1 235.308} C_DIS
LIN {X 0.009,Y -479.307,Z 1186.099,A 0.000,B 0.000,C 90.000,E1 233.783} C_DIS
LIN {X 0.061,Y -476.056,Z 1186.085,A 0.000,B 0.000,C 90.000,E1 231.295} C_DIS
LIN {X -0.221,Y -473.714,Z 1186.075,A 0.000,B 0.000,C 90.000,E1 229.461} C_DIS
LIN {X 0.189,Y -472.141,Z 1186.068,A 0.000,B 0.000,C 90.000,E1 228.162} C_DIS
LIN {X -0.197,Y -467.564,Z 1186.049,A 0.000,B 0.000,C 90.000,E1 224.757} C_DIS
LIN {X -0.218,Y -464.714,Z 1186.033,A 0.000,B 0.000,C 90.000,E1 221.919} C_DIS
LIN {X -0.294,Y -463.208,Z 1186.010,A 0.000,B 0.000,C 90.000,E1 217.810} C_DIS
LIN {X 0.259,Y -463.138,Z 1186.005,A 0.000,B 0.000,C 90.000,E1 216.790} C_DIS
LIN {X -0.056,Y -463.743,Z 1185.980,A 0.000,B 0.000,C 90.000,E1 212.388} C_DIS
LIN {X 0.286,Y -465.344,Z 1185.968,A 0.000,B 0.000,C 90.000,E1 210.129} C_DIS
LIN {X -0.100,Y -468.019,Z 1185.952,A 0.000,B 0.000,C 90.000,E1 207.334} C_DIS
LIN {X 0.142,Y -475.116,Z 1185.922,A 0.000,B 0.000,C 90.000,E1 201.972} C_DIS
LIN {X -0.211,Y -481.985,Z 1185.903,A 0.000,B 0.000,C 90.000,E1 198.598} C_DIS
LIN {X -0.163,Y -493.613,Z 1185.879,A 0.000,B 0.000,C 90.000,E1 194.300} C_DIS
LIN {X -0.098,Y -500.230,Z 1185.868,A 0.000,B 0.000,C 90.000,E1 192.175} C_DIS
LIN {X -0.017,Y -506.039,Z 1185.858,A 0.000,B 0.000,C 90.000,E1 190.366} C_DIS
LIN {X 0.110,Y -512.088,Z 1185.848,A 0.000,B 0.000,C 90.000,E1 188.568} C_DIS
LIN {X -0.185,Y -517.129,Z 1185.839,A 0.000,B 0.000,C 90.000,E1 187.125} C_DIS
LIN {X 0.129,Y -522.041,Z 1185.831,A 0.000,B 0.000,C 90.000,E1 185.625} C_DIS
LIN {X -0.035,Y -527.940,Z 1185.822,A 0.000,B 0.000,C 90.000,E1 183.898} C_DIS
LIN {X -0.114,Y -531.895,Z 1185.815,A 0.000,B 0.000,C 90.000,E1 182.751} C_DIS
LIN {X -0.140,Y -536.816,Z 1185.807,A 0.000,B 0.000,C 90.000,E1 181.318} C_DIS
LIN {X -0.039,Y -543.605,Z 1185.796,A 0.000,B 0.000,C 90.000,E1 179.312} C_DIS
LIN {X 0.200,Y -549.440,Z 1185.787,A 0.000,B 0.000,C 90.000,E1 177.593} C_DIS
LIN {X -0.053,Y -554.181,Z 1185.779,A 0.000,B 0.000,C 90.000,E1 176.216} C_DIS
LIN {X -0.189,Y -558.920,Z 1185.771,A 0.000,B 0.000,C 90.000,E1 174.837} C_DIS
LIN {X 0.054,Y -565.365,Z 1185.760,A 0.000,B 0.000,C 90.000,E1 172.875} C_DIS
LIN {X 0.179,Y -569.913,Z 1185.753,A 0.000,B 0.000,C 90.000,E1 171.489} C_DIS
LIN {X 0.079,Y -572.648,Z 1185.748,A 0.000,B 0.000,C 90.000,E1 170.679} C_DIS
LIN {X 0.054,Y -577.988,Z 1185.739,A 0.000,B 0.000,C 90.000,E1 169.050} C_DIS
LIN {X -0.079,Y -584.103,Z 1185.729,A 0.000,B 0.000,C 90.000,E1 167.173} C_DIS
LIN {X -0.253,Y -587.650,Z 1185.723,A 0.000,B 0.000,C 90.000,E1 166.117} C_DIS
LIN {X -0.290,Y -592.797,Z 1185.714,A 0.000,B 0.000,C 90.000,E1 164.519} C_DIS
LIN {X -0.059,Y -597.922,Z 1185.705,A 0.000,B 0.000,C 90.000,E1 162.906} C_DIS
LIN {X -0.189,Y -600.488,Z 1185.701,A 0.000,B 0.000,C 90.000,E1 162.127} C_DIS
LIN {X 0.097,Y -604.645,Z 1185.693,A 0.000,B 0.000,C 90.000,E1 160.786} C_DIS
LIN {X -0.316,Y -608.689,Z 1185.686,A 0.000,B 0.000,C 90.000,E1 159.518} C_DIS
LIN {X -0.138,Y -611.063,Z 1185.682,A 0.000,B 0.000,C 90.000,E1 158.720} C_DIS
LIN {X -0.009,Y -614.980,Z 1185.675,A 0.000,B 0.000,C 90.000,E1 157.411} C_DIS
LIN {X -0.070,Y -619.667,Z 1185.666,A 0.000,B 0.000,C 90.000,E1 155.869} C_DIS
LIN {X -0.101,Y -622.641,Z 1185.660,A 0.000,B 0.000,C 90.000,E1 154.845} C_DIS
LIN {X -0.070,Y -626.236,Z 1185.653,A 0.000,B 0.000,C 90.000,E1 153.563} C_DIS
LIN {X 0.023,Y -629.764,Z 1185.646,A 0.000,B 0.000,C 90.000,E1 152.281} C_DIS
LIN {X 0.164,Y -633.134,Z 1185.639,A 0.000,B 0.000,C 90.000,E1 151.001} C_DIS
LIN {X 0.107,Y -636.360,Z 1185.632,A 0.000,B 0.000,C 90.000,E1 149.744} C_DIS
LIN {X 0.100,Y -639.383,Z 1185.625,A 0.000,B 0.000,C 90.000,E1 148.486} C_DIS
LIN {X -0.116,Y -641.663,Z 1185.620,A 0.000,B 0.000,C 90.000,E1 147.502} C_DIS
LIN {X 0.308,Y -644.387,Z 1185.613,A 0.000,B 0.000,C 90.000,E1 146.215} C_DIS
LIN {X -0.244,Y -647.381,Z 1185.604,A 0.000,B 0.000,C 90.000,E1 144.769} C_DIS
LIN {X 0.011,Y -650.128,Z 1185.596,A 0.000,B 0.000,C 90.000,E1 143.256} C_DIS
LIN {X -0.116,Y -652.322,Z 1185.589,A 0.000,B 0.000,C 90.000,E1 142.029} C_DIS
LIN {X -0.279,Y -656.032,Z 1185.578,A 0.000,B 0.000,C 90.000,E1 140.070} C_DIS
LIN {X 0.057,Y -658.031,Z 1185.573,A 0.000,B 0.000,C 90.000,E1 139.057} C_DIS
LIN {X 0.413,Y -661.708,Z 1185.563,A 0.000,B 0.000,C 90.000,E1 137.310} C_DIS
LIN {X -0.114,Y -664.305,Z 1185.556,A 0.000,B 0.000,C 90.000,E1 136.134} C_DIS
LIN {X -0.135,Y -668.532,Z 1185.546,A 0.000,B 0.000,C 90.000,E1 134.190} C_DIS
LIN {X 0.001,Y -673.654,Z 1185.533,A 0.000,B 0.000,C 90.000,E1 132.000} C_DIS
LIN {X 0.188,Y -677.072,Z 1185.525,A 0.000,B 0.000,C 90.000,E1 130.539} C_DIS
LIN {X -0.032,Y -680.086,Z 1185.519,A 0.000,B 0.000,C 90.000,E1 129.358} C_DIS
LIN {X -0.019,Y -684.187,Z 1185.509,A 0.000,B 0.000,C 90.000,E1 127.684} C_DIS
LIN {X 0.080,Y -688.416,Z 1185.500,A 0.000,B 0.000,C 90.000,E1 126.011} C_DIS
LIN {X -0.427,Y -690.728,Z 1185.495,A 0.000,B 0.000,C 90.000,E1 125.105} C_DIS
LIN {X -0.300,Y -693.496,Z 1185.488,A 0.000,B 0.000,C 90.000,E1 123.913} C_DIS
LIN {X -0.169,Y -695.589,Z 1185.483,A 0.000,B 0.000,C 90.000,E1 122.959} C_DIS
LIN {X -0.353,Y -698.095,Z 1185.477,A 0.000,B 0.000,C 90.000,E1 121.799} C_DIS
LIN {X 0.091,Y -700.444,Z 1185.470,A 0.000,B 0.000,C 90.000,E1 120.590} C_DIS
LIN {X 0.222,Y -702.497,Z 1185.464,A 0.000,B 0.000,C 90.000,E1 119.411} C_DIS
LIN {X 0.105,Y -703.972,Z 1185.458,A 0.000,B 0.000,C 90.000,E1 118.487} C_DIS
LIN {X -0.329,Y -705.338,Z 1185.453,A 0.000,B 0.000,C 90.000,E1 117.590} C_DIS
LIN {X -0.083,Y -706.096,Z 1185.449,A 0.000,B 0.000,C 90.000,E1 116.873} C_DIS
LIN {X 0.145,Y -706.591,Z 1185.444,A 0.000,B 0.000,C 90.000,E1 115.924} C_DIS
LIN {X 0.098,Y -706.690,Z 1185.442,A 0.000,B 0.000,C 90.000,E1 115.463} C_DIS
LIN {X 0.040,Y -706.516,Z 1185.438,A 0.000,B 0.000,C 90.000,E1 114.771} C_DIS
LIN {X 0.332,Y -706.398,Z 1185.436,A 0.000,B 0.000,C 90.000,E1 114.515} C_DIS
LIN {X -0.019,Y -705.543,Z 1185.434,A 0.000,B 0.000,C 90.000,E1 114.079} C_DIS
LIN {X 0.270,Y -704.948,Z 1185.432,A 0.000,B 0.000,C 90.000,E1 113.823} C_DIS
LIN {X -0.088,Y -702.827,Z 1185.430,A 0.000,B 0.000,C 90.000,E1 113.387} C_DIS
LIN {X 0.051,Y -702.190,Z 1185.429,A 0.000,B 0.000,C 90.000,E1 113.259} C_DIS
LIN {X 0.191,Y -701.233,Z 1185.429,A 0.000,B 0.000,C 90.000,E1 113.131} C_DIS
LIN {X -0.074,Y -696.129,Z 1185.426,A 0.000,B 0.000,C 90.000,E1 112.695} C_DIS
LIN {X -0.130,Y -694.414,Z 1185.426,A 0.000,B 0.000,C 90.000,E1 112.589} C_DIS
LIN {X 0.082,Y -691.319,Z 1185.425,A 0.000,B 0.000,C 90.000,E1 112.461} C_DIS
LIN {X 0.193,Y -685.479,Z 1185.424,A 0.000,B 0.000,C 90.000,E1 112.280} C_DIS
LIN {X -0.043,Y -683.966,Z 1185.424,A 0.000,B 0.000,C 90.000,E1 112.280} C_DIS
LIN {X -0.048,Y -677.209,Z 1185.424,A 0.000,B 0.000,C 90.000,E1 112.259} C_DIS
LIN {X -0.086,Y -606.367,Z 1185.424,A 0.000,B 0.000,C 90.000,E1 112.259} C_DIS
LIN {X -0.112,Y -601.749,Z 1185.422,A 0.000,B 0.000,C 90.000,E1 111.950} C_DIS
LIN {X 0.304,Y -590.202,Z 1185.417,A 0.000,B 0.000,C 90.000,E1 110.972} C_DIS
LIN {X 0.187,Y -580.263,Z 1185.412,A 0.000,B 0.000,C 90.000,E1 110.194} C_DIS
LIN {X -0.253,Y -571.362,Z 1185.409,A 0.000,B 0.000,C 90.000,E1 109.577} C_DIS
LIN {X -0.274,Y -563.809,Z 1185.406,A 0.000,B 0.000,C 90.000,E1 109.033} C_DIS
LIN {X -0.040,Y -557.574,Z 1185.403,A 0.000,B 0.000,C 90.000,E1 108.544} C_DIS
LIN {X -0.165,Y -554.280,Z 1185.401,A 0.000,B 0.000,C 90.000,E1 108.181} C_DIS
LIN {X 0.172,Y -553.427,Z 1185.400,A 0.000,B 0.000,C 90.000,E1 108.000} C_DIS
LIN {X 0.167,Y -552.692,Z 1185.399,A 0.000,B 0.000,C 90.000,E1 107.819} C_DIS
LIN {X 0.146,Y -551.799,Z 1185.397,A 0.000,B 0.000,C 90.000,E1 107.402} C_DIS
LIN {X 0.222,Y -551.468,Z 1185.394,A 0.000,B 0.000,C 90.000,E1 106.804} C_DIS
LIN {X -0.044,Y -553.247,Z 1185.381,A 0.000,B 0.000,C 90.000,E1 104.592} C_DIS
LIN {X -0.222,Y -553.860,Z 1185.376,A 0.000,B 0.000,C 90.000,E1 103.772} C_DIS
LIN {X -0.171,Y -555.583,Z 1185.364,A 0.000,B 0.000,C 90.000,E1 101.535} C_DIS
LIN {X -0.021,Y -557.217,Z 1185.355,A 0.000,B 0.000,C 90.000,E1 99.849} C_DIS
LIN {X -0.110,Y -558.388,Z 1185.349,A 0.000,B 0.000,C 90.000,E1 98.746} C_DIS
LIN {X -0.186,Y -559.479,Z 1185.342,A 0.000,B 0.000,C 90.000,E1 97.644} C_DIS
LIN {X 0.301,Y -560.429,Z 1185.336,A 0.000,B 0.000,C 90.000,E1 96.486} C_DIS
LIN {X -0.212,Y -561.609,Z 1185.327,A 0.000,B 0.000,C 90.000,E1 94.878} C_DIS
LIN {X -0.127,Y -562.706,Z 1185.318,A 0.000,B 0.000,C 90.000,E1 93.212} C_DIS
LIN {X 0.074,Y -564.109,Z 1185.307,A 0.000,B 0.000,C 90.000,E1 91.260} C_DIS
LIN {X 0.164,Y -565.365,Z 1185.298,A 0.000,B 0.000,C 90.000,E1 89.599} C_DIS
LIN {X -0.156,Y -566.690,Z 1185.287,A 0.000,B 0.000,C 90.000,E1 87.707} C_DIS
LIN {X -0.003,Y -567.848,Z 1185.278,A 0.000,B 0.000,C 90.000,E1 86.045} C_DIS
LIN {X 0.087,Y -568.791,Z 1185.271,A 0.000,B 0.000,C 90.000,E1 84.666} C_DIS
LIN {X -0.203,Y -569.941,Z 1185.261,A 0.000,B 0.000,C 90.000,E1 83.053} C_DIS
LIN {X 0.063,Y -570.864,Z 1185.254,A 0.000,B 0.000,C 90.000,E1 81.659} C_DIS
LIN {X 0.168,Y -571.531,Z 1185.248,A 0.000,B 0.000,C 90.000,E1 80.557} C_DIS
LIN {X -0.088,Y -572.329,Z 1185.240,A 0.000,B 0.000,C 90.000,E1 79.218} C_DIS
LIN {X -0.146,Y -573.223,Z 1185.231,A 0.000,B 0.000,C 90.000,E1 77.589} C_DIS
LIN {X 0.057,Y -574.105,Z 1185.222,A 0.000,B 0.000,C 90.000,E1 75.936} C_DIS
LIN {X -0.276,Y -574.917,Z 1185.213,A 0.000,B 0.000,C 90.000,E1 74.338} C_DIS
LIN {X -0.064,Y -576.236,Z 1185.199,A 0.000,B 0.000,C 90.000,E1 71.873} C_DIS
LIN {X -0.002,Y -577.577,Z 1185.187,A 0.000,B 0.000,C 90.000,E1 69.699} C_DIS
LIN {X -0.046,Y -579.398,Z 1185.175,A 0.000,B 0.000,C 90.000,E1 67.539} C_DIS
LIN {X -0.068,Y -581.044,Z 1185.166,A 0.000,B 0.000,C 90.000,E1 65.921} C_DIS
LIN {X 0.048,Y -582.785,Z 1185.156,A 0.000,B 0.000,C 90.000,E1 64.024} C_DIS
LIN {X -0.058,Y -584.671,Z 1185.145,A 0.000,B 0.000,C 90.000,E1 62.153} C_DIS
LIN {X -0.006,Y -586.149,Z 1185.136,A 0.000,B 0.000,C 90.000,E1 60.539} C_DIS
LIN {X -0.032,Y -587.322,Z 1185.129,A 0.000,B 0.000,C 90.000,E1 59.203} C_DIS
LIN {X -0.035,Y -588.404,Z 1185.121,A 0.000,B 0.000,C 90.000,E1 57.867} C_DIS
LIN {X 0.291,Y -589.368,Z 1185.114,A 0.000,B 0.000,C 90.000,E1 56.501} C_DIS
LIN {X 0.145,Y -590.336,Z 1185.107,A 0.000,B 0.000,C 90.000,E1 55.182} C_DIS
LIN {X 0.012,Y -591.302,Z 1185.099,A 0.000,B 0.000,C 90.000,E1 53.863} C_DIS
LIN {X -0.045,Y -591.732,Z 1185.096,A 0.000,B 0.000,C 90.000,E1 53.336} C_DIS
LIN {X 0.370,Y -593.066,Z 1185.084,A 0.000,B 0.000,C 90.000,E1 51.170} C_DIS
LIN {X -0.065,Y -593.571,Z 1185.079,A 0.000,B 0.000,C 90.000,E1 50.150} C_DIS
LIN {X -0.351,Y -594.174,Z 1185.071,A 0.000,B 0.000,C 90.000,E1 48.852} C_DIS
LIN {X 0.235,Y -594.493,Z 1185.067,A 0.000,B 0.000,C 90.000,E1 48.000} C_DIS
LIN {X -0.243,Y -594.683,Z 1185.061,A 0.000,B 0.000,C 90.000,E1 46.986} C_DIS
LIN {X -0.105,Y -594.724,Z 1185.054,A 0.000,B 0.000,C 90.000,E1 45.648} C_DIS
LIN {X -0.169,Y -594.649,Z 1185.048,A 0.000,B 0.000,C 90.000,E1 44.595} C_DIS
LIN {X -0.237,Y -594.297,Z 1185.042,A 0.000,B 0.000,C 90.000,E1 43.542} C_DIS
LIN {X 0.349,Y -593.861,Z 1185.037,A 0.000,B 0.000,C 90.000,E1 42.690} C_DIS
LIN {X 0.069,Y -593.007,Z 1185.030,A 0.000,B 0.000,C 90.000,E1 41.391} C_DIS
LIN {X -0.196,Y -592.428,Z 1185.026,A 0.000,B 0.000,C 90.000,E1 40.620} C_DIS
LIN {X -0.262,Y -591.451,Z 1185.020,A 0.000,B 0.000,C 90.000,E1 39.564} C_DIS
LIN {X 0.113,Y -590.395,Z 1185.014,A 0.000,B 0.000,C 90.000,E1 38.463} C_DIS
LIN {X -0.092,Y -589.397,Z 1185.009,A 0.000,B 0.000,C 90.000,E1 37.684} C_DIS
LIN {X -0.024,Y -587.364,Z 1185.002,A 0.000,B 0.000,C 90.000,E1 36.343} C_DIS
LIN {X 0.067,Y -585.489,Z 1184.996,A 0.000,B 0.000,C 90.000,E1 35.264} C_DIS
LIN {X -0.001,Y -583.071,Z 1184.990,A 0.000,B 0.000,C 90.000,E1 34.199} C_DIS
LIN {X 0.029,Y -581.739,Z 1184.987,A 0.000,B 0.000,C 90.000,E1 33.658} C_DIS
LIN {X -0.109,Y -578.514,Z 1184.981,A 0.000,B 0.000,C 90.000,E1 32.594} C_DIS
